           ELSE  // 异常状态处理
               #状态 := 0;  // 恢复到停止状态
               #上阀控制 := FALSE;
               #下阀控制 := FALSE;
       END_CASE;

       // 更新输出状态
       #当前状态 := #状态;
END_FUNCTION_BLOCK

FUNCTION_BLOCK "四参数辅助"   // FB42, SCL
{ S7_Optimized_Access := 'TRUE' }
VERSION : 0.1
// stored: AutoNumber true, IsIECCheckEnabled false, IsRetainMemResEnabled false, MemoryReserve 100, SetENOAutomatically false, UDAEnableTagReadback false
   VAR_INPUT
      启动送风机 : Bool;   // 启动送风机命令
      关闭送风机 : Bool;   // 关闭送风机命令
      设定送风流量 : Real;   // 送风流量设定值
      实际送风流量 : Real;   // 流量变送器测量的实际流量
      流量上阈值 : Real := 10.0;   // 合格区间上限偏差值
      流量下阈值 : Real := 5.0;   // 合格区间下限偏差值
   END_VAR
   VAR_IN_OUT
      调节单元 : Real := 4.0;   // 频率调节单元 4Hz/时间
      调节时间 : Real := 30.0;   // 时间为秒
      调节时间PV : Real;
      变频器频率设定 : Real;   // 输出到变频器的频率设定
   END_VAR
   VAR
      运行状态 : Int := 0;   // 0: 停止, 1: 启动中, 2: 运行中, 3: 关闭中
      起始频率 : Real := 10.0;   // 起始频率10Hz
      最高频率 : Real := 50.0;   // 最高频率50Hz
      频率设定值 : Real := 0.0;   // 内部频率设定值
      流量合格 : Bool := FALSE;   // 流量是否在合格区间内
      TON1 : TON_TIME;
   END_VAR
BEGIN

       // 判断流量是否在合格区间内
       #流量合格 := (#实际送风流量 >= (#设定送风流量 - #流量下阈值)) AND
       (#实际送风流量 <= (#设定送风流量 + #流量上阈值));

       // 状态机
       CASE #运行状态 OF
           0:  // 停止状态
               IF #启动送风机 THEN
                   #运行状态 := 1;  // 转到启动状态
                   #频率设定值 := #起始频率;
                  // #送风机运行 := TRUE;
               END_IF;

           1:  // 启动状态
               IF #关闭送风机 THEN
                   #运行状态 := 3;  // 收到关闭命令，转到关闭状态
               ELSIF #流量合格 THEN
                   #运行状态 := 2;  // 流量达到合格区间，转到运行状态
               ELSIF #TON1.Q THEN
                   // 每分钟调整，最多增减4Hz
                   IF #实际送风流量 < #设定送风流量 - #流量下阈值 THEN
                       // 流量不足，增加频率
                       #频率设定值 := #频率设定值 + #调节单元;
                       IF #频率设定值 > #最高频率 THEN
                           #频率设定值 := #最高频率;
                       END_IF;
                   ELSIF #实际送风流量 > #设定送风流量 + #流量上阈值 THEN
                       // 流量过大，减少频率
                       #频率设定值 := #频率设定值 - #调节单元;
                       IF #频率设定值 < #起始频率 THEN
                           #频率设定值 := #起始频率;
                       END_IF;
                   END_IF;
               END_IF;

           2:  // 运行状态（流量稳定）
               IF #关闭送风机 THEN
                   #运行状态 := 3;  // 收到关闭命令，转到关闭状态
               ELSIF NOT #流量合格 AND #TON1.Q THEN
                   #运行状态 := 1;  // 流量不再合格，转回启动状态继续调节
               END_IF;

           3:  // 关闭状态
               IF #TON1.Q THEN
                   // 每分钟减少4Hz
                   #频率设定值 := #频率设定值 - #调节单元;

                   // 频率低于10Hz时关闭送风机
                   IF #频率设定值 < #起始频率 THEN
                     //  #送风机运行 := FALSE;
                       #频率设定值 := #起始频率;
                       #运行状态 := 0;  // 回到停止状态
                   END_IF;
               END_IF;
       END_CASE;

       #TON1(IN:=NOT #TON1.Q,
             PT:=DINT_TO_TIME(REAL_TO_DINT(#调节时间*1000)));

       #调节时间PV:=DINT_TO_REAL(TIME_TO_DINT(#TON1.ET))*1000;
       // 输出频率设定值
       #变频器频率设定 := #频率设定值;
END_FUNCTION_BLOCK

FUNCTION_BLOCK "闭式保压块"   // FB27, SCL
{ S7_Optimized_Access := 'TRUE' }
VERSION : 0.1
// stored: AutoNumber true, IsIECCheckEnabled false, IsRetainMemResEnabled false, MemoryReserve 100, SetENOAutomatically false, UDAEnableTagReadback false
   VAR_OUTPUT
      MBY等待保压 : Bool;
      MBY正在充气 : Bool;
      MBY保压不佳 : Bool;
      MBY正在保压 : Bool;
      MBY保压正常 : Bool;
   END_VAR
   VAR_IN_OUT
      模式设定 : Real;
      MBY保压 : Bool;
      MQT其他阀 : Bool;
      MCQ充气阀 : Bool;
      MCZ重置 : Bool;
      当前阶段 : Int;
      SV保压低设定 : Real;
      SV保压高设定 : Real;
      SV保压差值 : Real;
      SV保压时 : UInt;
      SV保压分 : UInt;
      SV保压秒 : UInt;
      PV塔内压力 { ExternalAccessible := 'False'; ExternalVisible := 'False'; ExternalWritable := 'False'} : Real;
      PV保压前 { ExternalAccessible := 'False'; ExternalVisible := 'False'; ExternalWritable := 'False'} : Real;
      PV保压后 { ExternalAccessible := 'False'; ExternalVisible := 'False'; ExternalWritable := 'False'} : Real;
      PV保压当前差值 { ExternalAccessible := 'False'; ExternalVisible := 'False'; ExternalWritable := 'False'} : Real;
      PV保压时 { ExternalAccessible := 'False'; ExternalVisible := 'False'; ExternalWritable := 'False'} : UInt;
      PV保压分 { ExternalAccessible := 'False'; ExternalVisible := 'False'; ExternalWritable := 'False'} : UInt;
      PV保压秒 { ExternalAccessible := 'False'; ExternalVisible := 'False'; ExternalWritable := 'False'} : UInt;
   END_VAR
   VAR
      T_1HZ { S7_SetPoint := 'True'} : TON_TIME;
      RT1 { S7_SetPoint := 'True'} : R_TRIG;
   END_VAR
BEGIN
   IF #模式设定 = 1.0 OR #模式设定 = 2.0  THEN

       #RT1(CLK := #MBY保压);
       IF #RT1.Q THEN
           #当前阶段 := 1;
       END_IF;
       IF #MBY保压 THEN
           IF #当前阶段 = 5 THEN
               #当前阶段 := 1;
           END_IF;
      ELSE
           #当前阶段 := 5; 
       END_IF;



       CASE #当前阶段 OF
           1://开始充气
               #MQT其他阀 := 0;
               #MCQ充气阀 := 1;
               #MBY等待保压 := 0;
               #MBY正在充气 := 1;
               #MBY保压不佳 := 0;
               #MBY正在保压 := 0;
               #MBY保压正常 := 0;

               IF (#PV塔内压力 >= #SV保压低设定) AND (#PV塔内压力 <= #SV保压高设定) THEN
                   #MCQ充气阀 := 0;
                   #PV保压前 := #PV塔内压力;
                   #当前阶段 := 2;
               END_IF;
           2://时间记录
               #MQT其他阀 := 0;
               #MCQ充气阀 := 0;
               IF #T_1HZ.Q THEN
                   #PV保压秒 += 1;
                   IF #PV保压秒 >= 60 THEN
                       #PV保压分 += 1;
                       #PV保压秒 := 0;
                       IF #PV保压分 >= 60 THEN
                           #PV保压时 += 1;
                           #PV保压分 := 0;
                       END_IF;
                   END_IF;
               END_IF;
               IF (#PV保压时 > #SV保压时) OR ((#PV保压时 = #SV保压时) AND (#PV保压分 > #SV保压分)) OR ((#PV保压时 = #SV保压时) AND (#PV保压分 = #SV保压分) AND (#PV保压秒 >= #SV保压秒)) THEN
                   #PV保压后 := #PV塔内压力;
                   #当前阶段 := 3;
               END_IF;

               #MBY等待保压 := 0;
               #MBY正在充气 := 0;
               #MBY保压不佳 := 0;
               #MBY正在保压 := 1;
               #MBY保压正常 := 0;

           3://保压结束
               #PV保压当前差值 := ABS(#PV保压前 - #PV保压后);
               #MBY保压正常 := #PV保压当前差值 < #SV保压差值;
               #MBY保压不佳 := NOT (#PV保压当前差值 < #SV保压差值);
               IF #MBY保压正常 OR #MBY保压不佳 THEN
                   #MBY正在保压 := 0;
                   #当前阶段 :=4;
               END_IF;
           4://停止保压，并记录数据



               #MBY正在充气 := 0;

               #MBY正在保压 := 0;



           5://清空数据
               #MCQ充气阀 := 0;
               #MBY保压 := 0;
               #PV保压前 := 0;
               #PV保压后 := 0;
               #PV保压时 := 0;
               #PV保压分 := 0;
               #PV保压秒 := 0;


               #MBY等待保压 := 1;
               #MBY正在充气 := 0;

               #MBY正在保压 := 0;
               #MBY保压正常 := 0;
               #MBY保压不佳 := 0;

               #PV保压当前差值 := 0.0;
       END_CASE;

      (* IF #MCZ重置 THEN
           #当前阶段 := 5;
           #MCZ重置 := FALSE;
       END_IF; *)


       #T_1HZ(IN := NOT #T_1HZ.Q,
              PT := T#1S);
   END_IF;
END_FUNCTION_BLOCK

FUNCTION_BLOCK "A14-阀反馈报警"   // FB20, SCL
{ S7_Optimized_Access := 'TRUE' }
VERSION : 0.1
// stored: AutoNumber true, IsIECCheckEnabled false, IsRetainMemResEnabled false, MemoryReserve 100, SetENOAutomatically false, UDAEnableTagReadback false
   VAR
      补氮阀 : "A8-阀开关报警";
      进氮阀 : "A8-阀开关报警";
      泄压阀 : "A8-阀开关报警";
      气流雾化阀 : "A8-阀开关报警";
      输送进风阀 : "A8-阀开关报警";
      开式排风隔断阀 : "A8-阀开关报警";
      闭式排风隔断阀 : "A8-阀开关报警";
      开式进风隔断阀 : "A8-阀开关报警";
      闭式进风隔断阀 : "A8-阀开关报警";
      一级冷却水阀 : "A8-阀开关报警";
      二级冷冻水阀 : "A8-阀开关报警";
      一级排液阀 : "A8-阀开关报警";
      二级排液阀 : "A8-阀开关报警";
      除雾排液阀 : "A8-阀开关报警";
      溶剂回收排放阀 : "A8-阀开关报警";
      进风冷却水阀 : "A8-阀开关报警";
      塔顶清洗球阀 : "A8-阀开关报警";
      清洗伸缩气缸 : "A8-阀开关报警";
      "71阀开关报警_Instance" { S7_SetPoint := 'True'} : "A8-阀开关报警";
      "71阀开关报警_Instance_1" { S7_SetPoint := 'True'} : "A8-阀开关报警";
   END_VAR
BEGIN

   #补氮阀(阀开报警 => "ABD补氮阀开报警",
        阀关报警 => "ABD补氮阀关报警",
        阀状态 :="QBD补氮阀",
        阀开信号 := "IBD补氮阀开反馈",
        阀关信号 := "IBD补氮阀关反馈");

   #进氮阀(阀开报警 => "AJD进氮阀开报警",
        阀关报警 => "AJD进氮阀关报警",
        阀状态 := "QJD进氮阀",
        阀开信号 := "IJD进氮阀开反馈",
        阀关信号 := "IJD进氮阀关反馈");


   #泄压阀(阀开报警 => "AXY泄压阀开报警",
        阀关报警 => "AXY泄压阀关报警",
        阀状态 := "QXY泄压阀",
        阀开信号 := "IXY泄压阀开反馈",
        阀关信号 := "IXY泄压阀关反馈");

   #气流雾化阀(阀开报警 => "AQL气流雾化阀开报警",
          阀关报警 => "AQL气流雾化阀关报警",
          阀状态 := "QQL气流雾化阀",
          阀开信号 := "IQL气流雾化阀开反馈",
          阀关信号 := "IQL气流雾化阀关反馈");

   #输送进风阀(阀开报警 => "ASS输送进风阀开报警",
          阀关报警 => "ASS输送进风阀关报警",
          阀状态 := "QSS输送进风阀",
          阀开信号 := "ISF输送进风阀开反馈",
          阀关信号 := "ISF输送进风阀关反馈");


   #开式排风隔断阀(阀开报警 => "AKS开式排风隔断阀开报警",
            阀关报警 => "AKS开式排风隔断阀关报警",
            阀状态 := "QKS开式排风隔断阀",
            阀开信号 := "IKS开式排风隔断阀开反馈",
            阀关信号 := "IKS开式排风隔断阀关反馈");

   #闭式排风隔断阀(阀开报警 => "ABS闭式排风隔断阀开报警",
            阀关报警 => "ABS闭式排风隔断阀关报警",
            阀状态 := "QBS闭式排风隔断阀",
            阀开信号 := "IBS闭式排风隔断阀开反馈",
            阀关信号 := "IBS闭式排风隔断阀关反馈");


   #开式进风隔断阀(阀开报警 => "AKS开式进风隔断阀开报警",
            阀关报警 => "AKS开式进风隔断阀关报警",
            阀状态 := "QKS开式进风隔断阀",
            阀开信号 := "IKS开式进风隔断阀开反馈",
            阀关信号 := "IKS开式进风隔断阀关反馈");

   #闭式进风隔断阀(阀开报警 => "ABS闭式进风隔断阀开报警",
            阀关报警 => "ABS闭式进风隔断阀关报警",
            阀状态 := "QBS闭式进风隔断阀",
            阀开信号 := "IBS闭式进风隔断阀开反馈",
            阀关信号 := "IBS闭式进风隔断阀关反馈");

   #一级冷却水阀(阀开报警 => "AYJ一级冷却水阀开报警",
           阀关报警 => "AYJ一级冷却水阀关报警",
           阀状态 := "QYJ一级冷却水阀",
           阀开信号 := "IYJ一级冷却水阀开反馈",
           阀关信号 := "IYJ一级冷却水阀关反馈");


   #二级冷冻水阀(阀开报警 => "AEJ二级冷冻水阀开报警",
           阀关报警 => "AEJ二级冷冻水阀关报警",
           阀状态 := "QEJ二级冷冻水阀",
           阀开信号 := "IEJ二级冷冻水阀开反馈",
           阀关信号 := "IEJ二级冷冻水阀关反馈");

   #一级排液阀(阀开报警 => "AYJ一级排液阀开报警",
          阀关报警 => "AYJ一级排液阀关报警",
          阀状态 := "QYJ一级排液阀",
          阀开信号 := "IYJ一级排液阀开反馈",
          阀关信号 := "IYJ一级排液阀关反馈");


   #二级排液阀(阀开报警 => "AEJ二级排液阀开报警",
          阀关报警 => "AEJ二级排液阀关报警",
          阀状态 := "QEJ二级排液阀",
          阀开信号 := "IEJ二级排液阀开反馈",
          阀关信号 := "IEJ二级排液阀关反馈");

   #除雾排液阀(阀开报警 => "ACW除雾排液阀开报警",
          阀关报警 => "ACW除雾排液阀关报警",
          阀状态 := "QCW除雾排液阀",
          阀开信号 := "ICW除雾排液阀开反馈",
          阀关信号 := "ICW除雾排液阀关反馈");

   #溶剂回收排放阀(阀开报警 => "ARJ溶剂回收排放阀开报警",
            阀关报警 => "ARJ溶剂回收排放阀关报警",
            阀状态 := "QRJ溶剂回收排放阀",
            阀开信号 := "IRJ溶剂回收排放阀开反馈",
            阀关信号 := "IRJ溶剂回收排放阀关反馈");


   #进风冷却水阀(阀开报警 => "AJF进风冷却水阀开报警",
           阀关报警 => "AJF进风冷却水阀关报警",
           阀状态 := "QJF进风冷却水阀",
           阀开信号 := "IJF进风冷却水阀开反馈",
           阀关信号 := "IJF进风冷却水阀关反馈");

   #塔顶清洗球阀(阀开报警 => "ATD塔顶清洗球阀开报警",
           阀关报警 => "ATD塔顶清洗球阀关报警",
           阀状态 := "QTD塔顶清洗球阀",
           阀开信号 := "ITD塔顶清洗球阀开反馈",
           阀关信号 := "ITD塔顶清洗球阀关反馈");


   (* #清洗伸缩气缸(阀开报警 => "AQX清洗伸缩气缸开报警",
           阀关报警 => "AQX清洗伸缩气缸关报警",
           阀状态 := "QQG气缸升降阀",
           阀开信号 := "IQX清洗伸缩气缸开反馈",
           阀关信号 := "IQX清洗伸缩气缸关反馈"); *)
END_FUNCTION_BLOCK

FUNCTION_BLOCK "D3-布袋记录"   // FB74, SCL
{ S7_Optimized_Access := 'TRUE' }
VERSION : 0.1
// stored: AutoNumber true, IsIECCheckEnabled false, IsRetainMemResEnabled false, MemoryReserve 100, SetENOAutomatically false, UDAEnableTagReadback false
   VAR_INPUT
      事件触发器 : Bool;
      清除日志 : Bool;
   END_VAR
   VAR_IN_OUT
      事件记录 : Array[1..20] of String[20];
      事件编号 : Array[1..20] of Int;
      当前记录次数 : Int;
   END_VAR
   VAR
      R_TRIG_Instance { S7_SetPoint := 'True'} : R_TRIG;
      tm_DTL { ExternalAccessible := 'False'; ExternalVisible := 'False'; ExternalWritable := 'False'} : DTL;
   END_VAR
   VAR_TEMP
      tm_Ret : Int;
      tm_i : Int;
      tm_str : String[20];
      tm_year : String[5];
      tm_month : String[3];
      tm_day : String[3];
      tm_hour : String[3];
      tm_minute : String[3];
      tm_second : String[3];
      tm_strcount : String[5];
      tm_strC : String[4];
      tm_empty : Array[1..20] of String[20];
      tm_cempty : Array[1..20] of Int;
   END_VAR
BEGIN
   #R_TRIG_Instance(CLK:=#事件触发器);
   IF #当前记录次数 < 1 THEN
       #当前记录次数 := 1;
   END_IF;

   IF (#当前记录次数 > 9999) OR  #清除日志 THEN
       #当前记录次数 := 1;

       #事件记录 := #tm_empty;
       #事件编号 := #tm_cempty;
       #当前记录次数 := 1;
   END_IF;

   IF #R_TRIG_Instance.Q THEN
       #tm_Ret := RD_LOC_T(#tm_DTL);
       #tm_year := UINT_TO_STRING(#tm_DTL.YEAR);
       #tm_month := USINT_TO_STRING(#tm_DTL.MONTH);
       #tm_day := USINT_TO_STRING(#tm_DTL.DAY);
       #tm_hour := USINT_TO_STRING(#tm_DTL.HOUR+7);
       #tm_minute := USINT_TO_STRING(#tm_DTL.MINUTE);
       #tm_second := USINT_TO_STRING(#tm_DTL.SECOND);
       #tm_str := '';
       #tm_str[1] := #tm_year[2];
       #tm_str[2] := #tm_year[3];
       #tm_str[3] := #tm_year[4];
       #tm_str[4] := #tm_year[5];
       #tm_str[5] := '-';
       IF LEN(#tm_month) = 3 THEN
           #tm_str[6] := #tm_month[2];
           #tm_str[7] := #tm_month[3];
       ELSE
           #tm_str[6] := '0';
           #tm_str[7] := #tm_month[2];
       END_IF;
       #tm_str[8] := '-';
       IF LEN(#tm_day)= 3 THEN
       #tm_str[9] := #tm_day[2];
       #tm_str[10] := #tm_day[3];
   ELSE
       #tm_str[9] := '0';
       #tm_str[10] := #tm_day[2];;
   END_IF;

   #tm_str[11] := ' ';
   IF LEN(#tm_hour) = 3 THEN
       #tm_str[12] := #tm_hour[2];
       #tm_str[13] := #tm_hour[3];
   ELSE
       #tm_str[12] := '0';
       #tm_str[13] := #tm_hour[2];
   END_IF;
   #tm_str[14] := ':';
   IF LEN(#tm_minute) = 3 THEN
       #tm_str[15] := #tm_minute[2];
       #tm_str[16] := #tm_minute[3];
   ELSE
       #tm_str[15] := '0';
       #tm_str[16] := #tm_minute[2];
   END_IF;
       #tm_str[17] := ':';
       IF LEN(#tm_second) = 3 THEN
           #tm_str[18] := #tm_second[2];
           #tm_str[19] := #tm_second[3];
       ELSE
           #tm_str[18] := '0';
           #tm_str[19] := #tm_second[2];
       END_IF;
       #tm_strcount := INT_TO_STRING(#当前记录次数);
       IF LEN(#tm_strcount) = 2 THEN
           #tm_strC[1] := '0';
           #tm_strC[2] := '0';
           #tm_strC[3] := '0';
           #tm_strC[4] := #tm_strcount[2];
       END_IF;

       IF LEN(#tm_strcount) = 3 THEN
           #tm_strC[1] := '0';
           #tm_strC[2] := '0';
           #tm_strC[3] := #tm_strcount[2];
           #tm_strC[4] := #tm_strcount[3];
       END_IF;
       IF LEN(#tm_strcount) = 4 THEN
           #tm_strC[1] := '0';
           #tm_strC[2] := #tm_strcount[2];
           #tm_strC[3] := #tm_strcount[3];
           #tm_strC[4] := #tm_strcount[4];
       END_IF;
       IF LEN(#tm_strcount) =5 THEN
           #tm_strC[1] := #tm_strcount[2];
           #tm_strC[2] := #tm_strcount[3];
           #tm_strC[3] := #tm_strcount[4];
           #tm_strC[4] := #tm_strcount[5];
       END_IF;



       IF #当前记录次数 < 20 THEN
           #事件记录[#当前记录次数] := #tm_str;
           #事件编号[#当前记录次数] :=#当前记录次数;
       ELSE
           FOR #tm_i := 1 TO 19 DO
               #事件编号[#tm_i] := #事件编号[#tm_i + 1];
               #事件编号[#tm_i] := #事件编号[#tm_i + 1];
           END_FOR;
           #事件记录[20] := #tm_str;
           #事件编号[20] := #当前记录次数;
       END_IF;
       #当前记录次数 := #当前记录次数 + 1;
   END_IF;
END_FUNCTION_BLOCK

FUNCTION_BLOCK "12放空阀"   // FB8, SCL
{ S7_Optimized_Access := 'FALSE' }
VERSION : 0.1
// stored: AutoNumber true, IsIECCheckEnabled false, SetENOAutomatically false, UDAEnableTagReadback false
   VAR_INPUT
      条件1 : Real;
      工程上限 : Real;
      工程下限 : Real;
      模拟高限 : Int;
      模拟低限 : Int;
   END_VAR
   VAR_IN_OUT
      模式设定 : Real;
      阀门启动 : Bool;
      阀门输出 : Bool;
      百分比设定值 : Real;
      输出百分比 : Int;
      PID反馈模拟量 : Int;
      YS映射到阀开度 : Real;
   END_VAR
   VAR DB_SPECIFIC
      动画 : Int;
      ST1 : Real;
   END_VAR
   VAR_TEMP
      TEMP_1 : Int;
   END_VAR
BEGIN
   // "IEC_Timer_0_DB".TON(IN:=#输出电源开,
   //                      PT:=T#10s,
   //                      Q=>  #阀开报警检测位);
   // IF #阀开报警检测位 AND #阀开信号  THEN
   //     #阀开异常报警 := TRUE;
   // ELSE
   //     #阀开异常报警 := FALSE;
   // END_IF;
   // "IEC_Timer_0_DB_1".TON (IN:=NOT #输出电源开,
   //                        PT:=T#10s,
   //                        Q=>#阀关报警检测位);
   // IF #阀关报警检测位 AND #阀关信号  THEN
   //     #阀关异常报警 := TRUE; ELSE
   //     #阀关异常报警 :=FALSE;
   // END_IF;
   //手动控制--------------------------------------------------------------------------------------------------------------
   IF #模式设定 = 2.0 THEN

       IF #阀门启动 THEN
           #阀门输出 := TRUE;
           #输出百分比 := REAL_TO_INT((#百分比设定值 - #工程下限) * (#模拟高限 - #模拟低限) / (#工程上限 - #工程下限) + #模拟低限);

       END_IF;
       IF NOT #阀门启动 THEN
           #阀门输出 := FALSE;
           #输出百分比 := REAL_TO_INT(#工程下限);

       END_IF;

   END_IF;

   // 自动启动--------------------------------------------------------------------------------------------------------------
   IF #阀门输出 AND #模式设定 = 1.0 THEN
       (* #输出百分比 := REAL_TO_INT((#百分比设定值 - #工程下限) * (#模拟高限 - #模拟低限) / (#工程上限 - #工程下限) + #模拟低限); *)


       #ST1 := NORM_X_REAL(MIN := 5530, VALUE := #输出百分比, MAX := 27648);
       #YS映射到阀开度 := SCALE_X_REAL(MIN := 0, VALUE := #ST1, MAX := 100);


   END_IF;
   IF NOT #阀门输出 THEN
       #YS映射到阀开度 := 0;
   END_IF;




   (* #TON1(IN := #电机输出 AND #电机电流 < 10,
                          PT := T#60s,
                          Q => #P1);

   IF #P1 OR #电机报警信号 THEN
       #电机报警输出 := TRUE;
   ELSE
       #电机报警输出 := FALSE;
   END_IF; *)



   IF #阀门输出  THEN
       IF "Clock_1Hz" THEN
           #TEMP_1 := #TEMP_1 + 1;
       END_IF;

       IF #TEMP_1 >= 3 THEN
           #TEMP_1 := 0;
       END_IF;
       IF #TEMP_1 < 1 THEN
           #动画 := 0;
       ELSE
           #动画 := 1;
       END_IF;

   END_IF;
   IF NOT #阀门输出 THEN
       #动画 := 0;
   END_IF;




   // IF #阀开异常报警 THEN
   //     #输出电源开 := FALSE;
   // END_IF;
   // IF #阀关异常报警 THEN
   //     #输出电源开 := TRUE;
   // END_IF;
END_FUNCTION_BLOCK

FUNCTION_BLOCK "21模拟量输入"   // FB2, SCL
{ S7_Optimized_Access := 'TRUE' }
VERSION : 0.1
// stored: AutoNumber true, IsIECCheckEnabled false, IsRetainMemResEnabled false, MemoryReserve 100, SetENOAutomatically false, UDAEnableTagReadback false
   VAR_INPUT
      HMI上限 : Real;
      HMI下限 : Real;
      PLC上限 : Int := 27648;
      PLC下限 : Int;
   END_VAR
   VAR_IN_OUT
      "PLC-仪表" : Int;
      HMI仪表 : Real;
   END_VAR
   VAR
      DBD28 : Real;
   END_VAR
BEGIN
   #DBD28 := NORM_X_REAL(MIN := #PLC下限, VALUE := #"PLC-仪表", MAX := #PLC上限);
   #HMI仪表 := SCALE_X_REAL(MIN := #HMI下限, VALUE := #DBD28, MAX := #HMI上限);
END_FUNCTION_BLOCK

FUNCTION_BLOCK "22模拟量输入修正"   // FB10, SCL
{ S7_Optimized_Access := 'TRUE' }
VERSION : 0.1
// stored: AutoNumber true, IsIECCheckEnabled false, IsRetainMemResEnabled false, MemoryReserve 100, SetENOAutomatically false, UDAEnableTagReadback false
   VAR_INPUT
      设备启动 : Bool;
      HMI上限 : Real;
      HMI下限 : Real;
      PLC上限 : Int := 27648;
      PLC下限 : Int;
   END_VAR
   VAR_IN_OUT
      "PLC-仪表" : Int;
      HMI仪表 : Real;
   END_VAR
   VAR
      DBD1 : Real;
   END_VAR
BEGIN
   IF #设备启动 THEN

   #DBD1 := NORM_X_REAL(MIN := #PLC下限, VALUE := #"PLC-仪表", MAX := #PLC上限);
   #HMI仪表 := SCALE_X_REAL(MIN := #HMI下限, VALUE := #DBD1, MAX := #HMI上限);

   ELSE

       #HMI仪表 := 0;
   END_IF;
END_FUNCTION_BLOCK

FUNCTION_BLOCK "23模拟量输出"   // FB36, SCL
{ S7_Optimized_Access := 'TRUE' }
VERSION : 0.1
// stored: AutoNumber true, IsIECCheckEnabled false, IsRetainMemResEnabled false, MemoryReserve 100, SetENOAutomatically false, UDAEnableTagReadback false
   VAR_INPUT
      HMI上限 : Real;
      HMI下限 : Real;
      PLC上限 : Int;
      PLC下限 : Int;
   END_VAR
   VAR_IN_OUT
      PLC调控 : Int;
      HMI设定 : Real;
   END_VAR
   VAR
      DBD1 : Real;
   END_VAR
BEGIN
   #DBD1 := NORM_X_REAL(MIN := #HMI下限, VALUE := #HMI设定, MAX := #HMI上限);
   #PLC调控 := SCALE_X_INT(MIN := #PLC下限, VALUE := #DBD1, MAX := #PLC上限);
END_FUNCTION_BLOCK

FUNCTION_BLOCK "24模拟量其他"   // FB4, SCL
{ S7_Optimized_Access := 'TRUE' }
VERSION : 0.1
// stored: AutoNumber true, IsIECCheckEnabled false, IsRetainMemResEnabled false, MemoryReserve 100, SetENOAutomatically false, UDAEnableTagReadback false
BEGIN
END_FUNCTION_BLOCK

FUNCTION_BLOCK "30-加热控制"   // FB17, SCL
{ S7_Optimized_Access := 'TRUE' }
VERSION : 0.1
// stored: AutoNumber true, IsIECCheckEnabled false, IsRetainMemResEnabled false, MemoryReserve 100, SetENOAutomatically false, UDAEnableTagReadback false
   VAR_INPUT
      条件1 : Real;
   END_VAR
   VAR_IN_OUT
      模式设定 : Real;
      加热控制按钮 : Bool;
      电力调整器信号 : Bool;
      电力调整器报警 : Bool;
      机械温报警信号 : Bool;
      循环风机反馈 : Real;
      循环风机 : Bool;
      加热输出 : Bool;
      AO : Int;
      安全停机 : Bool;
   END_VAR
BEGIN

   //手动控制--------------------------------------------------------------------------------------------------------------
   IF #模式设定 = 2.0 THEN
       //预热器加热手动控制
       IF #加热控制按钮
           AND #电力调整器报警 = FALSE AND #机械温报警信号 = FALSE AND #循环风机反馈 > 20 AND #循环风机 THEN
           #加热输出 := TRUE;

       ELSE

           #加热输出 := FALSE;

       END_IF;
   END_IF;
   IF #模式设定 = 2.0  THEN
       //预热器加热手动控制
       IF NOT #加热控制按钮 THEN


           #加热输出 := FALSE;

       END_IF;
   END_IF;

   //自动模式
   IF #加热输出 THEN
       #AO := -256;
   END_IF;


   IF NOT #加热输出 THEN
       #AO := 0;
   END_IF;
   IF #电力调整器信号 THEN
       #电力调整器报警 := TRUE;
   ELSE


       #电力调整器报警 := FALSE;
   END_IF;

   IF
       #模式设定 = 1 AND (#电力调整器报警 OR #机械温报警信号) THEN

       #安全停机 := 1;
   END_IF;
END_FUNCTION_BLOCK

FUNCTION_BLOCK "31-温度控制"   // FB21, LAD
{ S7_Optimized_Access := 'FALSE' }
VERSION : 0.1
// stored: AutoNumber true, IsIECCheckEnabled false, SetENOAutomatically false, UDAEnableTagReadback false
   VAR_IN_OUT
      进温设定 : Real;
      加热器开关 : Bool;
      自整定开关 : Bool;
      进温读 : Real;
      出温读 : Real;
      尾温读 : Real;
      进风温度P : Real;
      进风温度I : Real;
      进风温度D : Real;
      JF进风温度写读 : Real;
   END_VAR
   VAR DB_SPECIFIC
      CTU { S7_SetPoint := 'True'} : CTU_INT;
      TEMP { S7_SetPoint := 'True'} : Bool;
      TP : Array[0..40] of Bool;
      T1_PV_读 : Int;
      T2_PV_读 : Int;
      T3_PV_读 : Int;
      T4_PV_读 : Int;
      T5_PV_读 : Int;
      T1_SV_写 : Int;
      T1_P值比对1 : Int;
      T1_P值比对2 : Int;
      ST1 : Real;
      ST2 : Real;
      ST3 : Real;
      ST4 : Real;
      ST5 : Real;
      ST16 : Real;
      ST17 : Real;
      ST18 : Real;
      ST20 : Real;
      ST21 : Real;
      ST22 : Real;
      进温P读 : Int;
      进温I读 : Int;
      进温D读 : Int;
      T1_P_I_D_读 : Array[0..2] of Int;
      IEC_Timer_0_Instance { S7_SetPoint := 'True'} : TON_TIME;
      JF进风温度写读辅 { S7_SetPoint := 'True'} : Int;
      进温AT_写 : Int;
      进温AT_读 : Int;
      自整定开关字 : Int;
      加热器开关字 : Int;
   END_VAR
   VAR
      Modbus_Comm_Load_Instance { S7_SetPoint := 'True'} : Modbus_Comm_Load;
      Modbus_Master { S7_SetPoint := 'True'} : Modbus_Master;
   END_VAR
   VAR_TEMP   // added for the SCL form of the ladder/FBD networks
      _w1 : Bool;
      _w2 : Bool;
      _w3 : Bool;
      _w4 : Bool;
   END_VAR
BEGIN

REGION Network 1
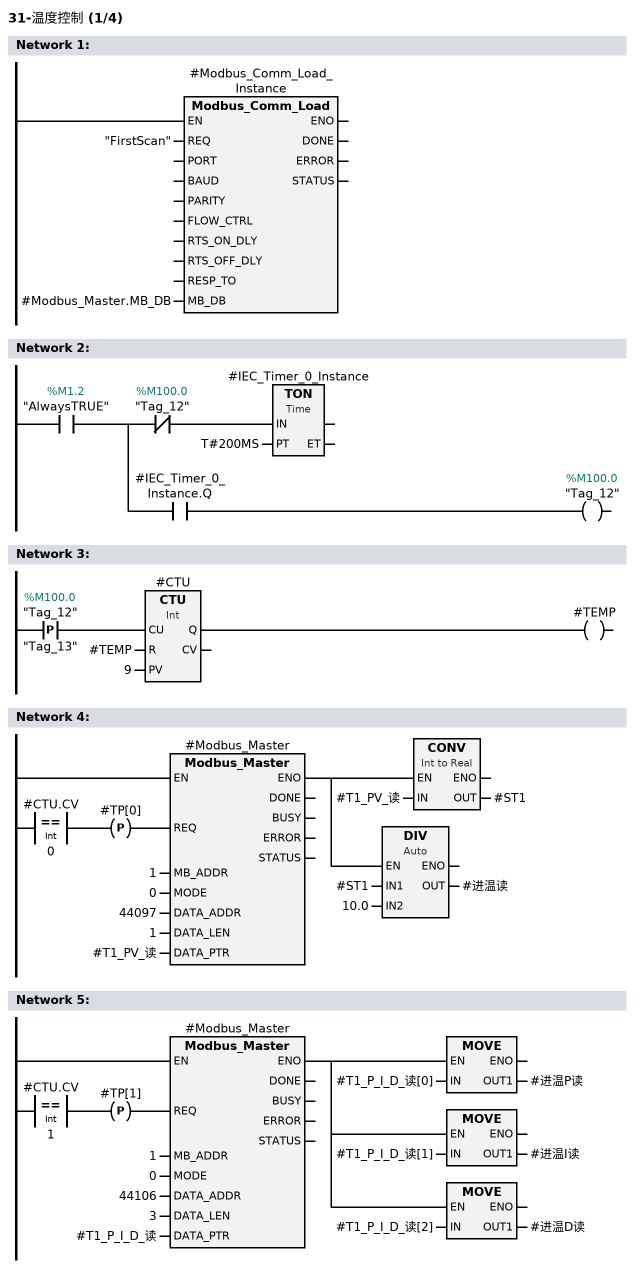
   RUNG wire#powerrail
      #Modbus_Comm_Load_Instance.Modbus_Comm_Load(REQ := "FirstScan", PORT :=, BAUD :=, PARITY :=, FLOW_CTRL :=, RTS_ON_DLY :=, RTS_OFF_DLY :=, RESP_TO :=, MB_DB := #Modbus_Master.MB_DB, DONE =>, ERROR =>, STATUS =>)
   END_RUNG
   // the same network as SCL:
   #Modbus_Comm_Load_Instance(REQ := "FirstScan", MB_DB := #Modbus_Master.MB_DB);   // Modbus_Comm_Load
END_REGION

REGION Network 2
   RUNG wire#powerrail
      Contact( "AlwaysTRUE" )
      wire#w1
      I_Contact( "Tag_12" )
      { S7_Templates := "time_type := Time" } #IEC_Timer_0_Instance.TON(pt := T#200MS, et =>)
   END_RUNG
   RUNG wire#w1
      Contact( #IEC_Timer_0_Instance.Q )
      Coil( "Tag_12" )
   END_RUNG
   // the same network as SCL:
   #IEC_Timer_0_Instance(IN := "AlwaysTRUE" AND NOT "Tag_12", PT := T#200MS);   // TON
   "Tag_12" := "AlwaysTRUE" AND #IEC_Timer_0_Instance.Q;
END_REGION

REGION Network 3
   RUNG wire#powerrail
      P_Contact(operand := "Tag_12", bit := "Tag_13")
      { S7_Templates := "value_type := Int" } #CTU.CTU(r := #TEMP, pv := 9, cv =>)
      Coil( #TEMP )
   END_RUNG
   // the same network as SCL:
   #_w1 := "Tag_12" AND NOT "Tag_13";   // rising edge of "Tag_12"
   "Tag_13" := "Tag_12";
   #CTU(CU := #_w1, R := #TEMP, PV := 9);   // CTU
   #TEMP := #CTU.Q;
END_REGION

REGION Network 4
   RUNG wire#powerrail
      #Modbus_Master.Modbus_Master(REQ := wire#w1, MB_ADDR := 1, MODE := 0, DATA_ADDR := 44097, DATA_LEN := 1, DATA_PTR := #T1_PV_读, DONE =>, BUSY =>, ERROR =>, STATUS =>)
      wire#w2
      { S7_Templates := "[SrcType := Int, DestType := Real]" } Convert(in := #T1_PV_读, out => #ST1)
   END_RUNG
   RUNG wire#powerrail
      { S7_Templates := "SrcType := Int" } EQ_Contact(in1 := #CTU.CV, in2 := 0)
      P_Trig( #TP[0] )
   END_RUNG wire#w1
   RUNG wire#w2
      Div(in1 := #ST1, in2 := 10.0, out => #进温读)
   END_RUNG
   // the same network as SCL:
   #_w1 := #CTU.CV = 0;
   #_w2 := #_w1 AND NOT #TP[0];   // rising edge
   #TP[0] := #_w1;
   #Modbus_Master(REQ := #_w2,   // Modbus_Master
                  MB_ADDR := 1,
                  MODE := 0,
                  DATA_ADDR := 44097,
                  DATA_LEN := 1,
                  DATA_PTR := #T1_PV_读,
                  ENO => #_w3);
   IF #_w3 THEN
       #ST1 := INT_TO_REAL(#T1_PV_读);
       #进温读 := #ST1 / 10.0;
   END_IF;
END_REGION

REGION Network 5
   RUNG wire#powerrail
      #Modbus_Master.Modbus_Master(REQ := wire#w1, MB_ADDR := 1, MODE := 0, DATA_ADDR := 44106, DATA_LEN := 3, DATA_PTR := #T1_P_I_D_读, DONE =>, BUSY =>, ERROR =>, STATUS =>)
      wire#w2
      Move(in := #T1_P_I_D_读[0], out1 => #进温P读)
   END_RUNG
   RUNG wire#powerrail
      { S7_Templates := "SrcType := Int" } EQ_Contact(in1 := #CTU.CV, in2 := 1)
      P_Trig( #TP[1] )
   END_RUNG wire#w1
   RUNG wire#w2
      Move(in := #T1_P_I_D_读[1], out1 => #进温I读)
   END_RUNG
   RUNG wire#w2
      Move(in := #T1_P_I_D_读[2], out1 => #进温D读)
   END_RUNG
   // the same network as SCL:
   #_w1 := #CTU.CV = 1;
   #_w2 := #_w1 AND NOT #TP[1];   // rising edge
   #TP[1] := #_w1;
   #Modbus_Master(REQ := #_w2,   // Modbus_Master
                  MB_ADDR := 1,
                  MODE := 0,
                  DATA_ADDR := 44106,
                  DATA_LEN := 3,
                  DATA_PTR := #T1_P_I_D_读,
                  ENO => #_w3);
   IF #_w3 THEN
       #进温P读 := #T1_P_I_D_读[0];
       #进温I读 := #T1_P_I_D_读[1];
       #进温D读 := #T1_P_I_D_读[2];
   END_IF;
END_REGION

REGION Network 6
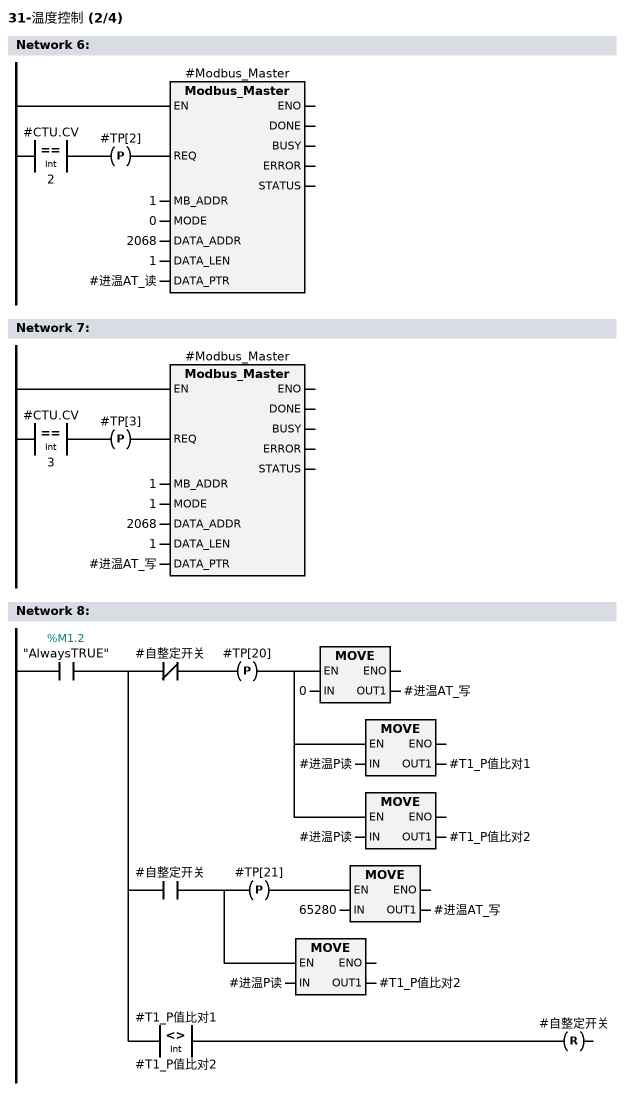
   RUNG wire#powerrail
      #Modbus_Master.Modbus_Master(REQ := wire#w1, MB_ADDR := 1, MODE := 0, DATA_ADDR := 2068, DATA_LEN := 1, DATA_PTR := #进温AT_读, DONE =>, BUSY =>, ERROR =>, STATUS =>)
   END_RUNG
   RUNG wire#powerrail
      { S7_Templates := "SrcType := Int" } EQ_Contact(in1 := #CTU.CV, in2 := 2)
      P_Trig( #TP[2] )
   END_RUNG wire#w1
   // the same network as SCL:
   #_w1 := #CTU.CV = 2;
   #_w2 := #_w1 AND NOT #TP[2];   // rising edge
   #TP[2] := #_w1;
   #Modbus_Master(REQ := #_w2, MB_ADDR := 1, MODE := 0, DATA_ADDR := 2068, DATA_LEN := 1, DATA_PTR := #进温AT_读);   // Modbus_Master
END_REGION

REGION Network 7
   RUNG wire#powerrail
      #Modbus_Master.Modbus_Master(REQ := wire#w1, MB_ADDR := 1, MODE := 1, DATA_ADDR := 2068, DATA_LEN := 1, DATA_PTR := #进温AT_写, DONE =>, BUSY =>, ERROR =>, STATUS =>)
   END_RUNG
   RUNG wire#powerrail
      { S7_Templates := "SrcType := Int" } EQ_Contact(in1 := #CTU.CV, in2 := 3)
      P_Trig( #TP[3] )
   END_RUNG wire#w1
   // the same network as SCL:
   #_w1 := #CTU.CV = 3;
   #_w2 := #_w1 AND NOT #TP[3];   // rising edge
   #TP[3] := #_w1;
   #Modbus_Master(REQ := #_w2, MB_ADDR := 1, MODE := 1, DATA_ADDR := 2068, DATA_LEN := 1, DATA_PTR := #进温AT_写);   // Modbus_Master
END_REGION

REGION Network 8
   RUNG wire#powerrail
      Contact( "AlwaysTRUE" )
      wire#w1
      I_Contact( #自整定开关 )
      P_Trig( #TP[20] )
      wire#w2
      Move(in := 0, out1 => #进温AT_写)
   END_RUNG
   RUNG wire#w2
      Move(in := #进温P读, out1 => #T1_P值比对1)
   END_RUNG
   RUNG wire#w2
      Move(in := #进温P读, out1 => #T1_P值比对2)
   END_RUNG
   RUNG wire#w1
      Contact( #自整定开关 )
      wire#w3
      P_Trig( #TP[21] )
      Move(in := 65280, out1 => #进温AT_写)
   END_RUNG
   RUNG wire#w3
      Move(in := #进温P读, out1 => #T1_P值比对2)
   END_RUNG
   RUNG wire#w1
      { S7_Templates := "SrcType := Int" } NE_Contact(in1 := #T1_P值比对1, in2 := #T1_P值比对2)
      R_Coil( #自整定开关 )
   END_RUNG
   // the same network as SCL:
   #_w1 := "AlwaysTRUE" AND NOT #自整定开关;
   #_w2 := #_w1 AND NOT #TP[20];   // rising edge
   #TP[20] := #_w1;
   IF #_w2 THEN
       #进温AT_写 := 0;
       #T1_P值比对1 := #进温P读;
       #T1_P值比对2 := #进温P读;
   END_IF;
   #_w3 := "AlwaysTRUE" AND #自整定开关;
   #_w4 := #_w3 AND NOT #TP[21];   // rising edge
   #TP[21] := #_w3;
   IF #_w4 THEN #进温AT_写 := 65280; END_IF;
   IF #_w3 THEN #T1_P值比对2 := #进温P读; END_IF;
   IF "AlwaysTRUE" AND (#T1_P值比对1 <> #T1_P值比对2) THEN #自整定开关 := FALSE; END_IF;
END_REGION

REGION Network 9
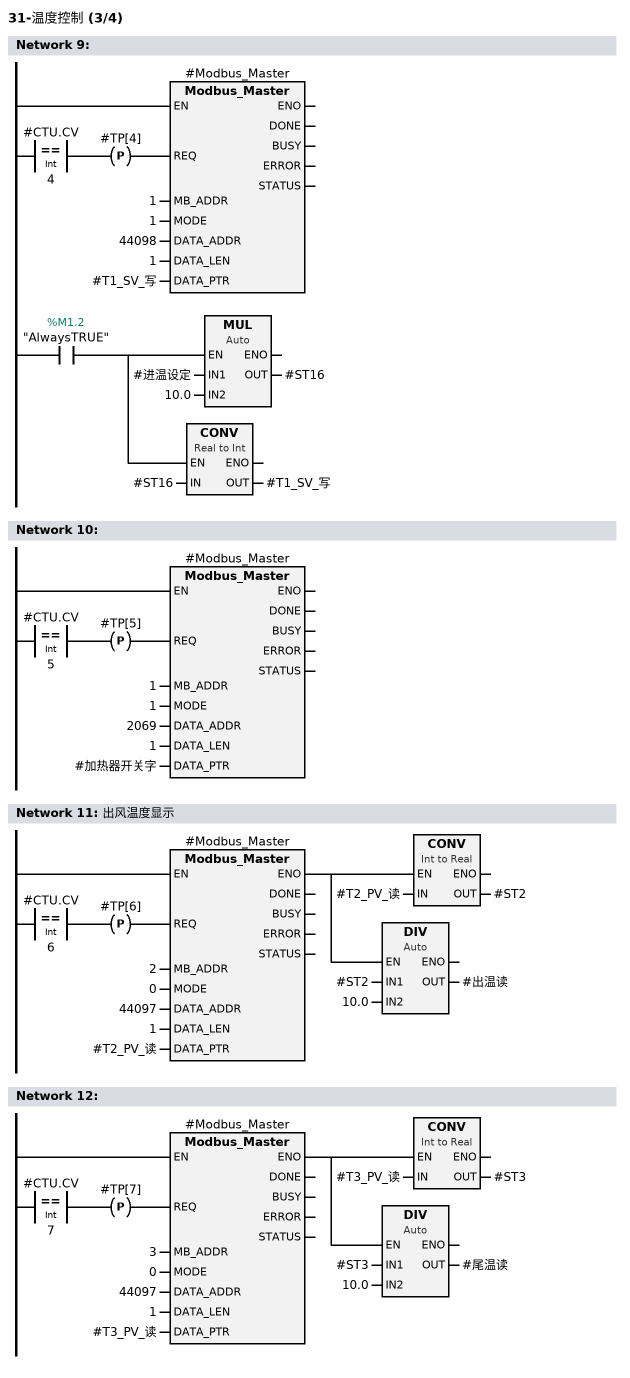
   RUNG wire#powerrail
      #Modbus_Master.Modbus_Master(REQ := wire#w1, MB_ADDR := 1, MODE := 1, DATA_ADDR := 44098, DATA_LEN := 1, DATA_PTR := #T1_SV_写, DONE =>, BUSY =>, ERROR =>, STATUS =>)
   END_RUNG
   RUNG wire#powerrail
      { S7_Templates := "SrcType := Int" } EQ_Contact(in1 := #CTU.CV, in2 := 4)
      P_Trig( #TP[4] )
   END_RUNG wire#w1
   RUNG wire#powerrail
      Contact( "AlwaysTRUE" )
      wire#w2
      Mul(in1 := #进温设定, in2 := 10.0, out => #ST16)
   END_RUNG
   RUNG wire#w2
      { S7_Templates := "[SrcType := Real, DestType := Int]" } Convert(in := #ST16, out => #T1_SV_写)
   END_RUNG
   // the same network as SCL:
   #_w1 := #CTU.CV = 4;
   #_w2 := #_w1 AND NOT #TP[4];   // rising edge
   #TP[4] := #_w1;
   #Modbus_Master(REQ := #_w2, MB_ADDR := 1, MODE := 1, DATA_ADDR := 44098, DATA_LEN := 1, DATA_PTR := #T1_SV_写);   // Modbus_Master
   IF "AlwaysTRUE" THEN
       #ST16 := #进温设定 * 10.0;
       #T1_SV_写 := REAL_TO_INT(#ST16);
   END_IF;
END_REGION

REGION Network 10
   RUNG wire#powerrail
      #Modbus_Master.Modbus_Master(REQ := wire#w1, MB_ADDR := 1, MODE := 1, DATA_ADDR := 2069, DATA_LEN := 1, DATA_PTR := #加热器开关字, DONE =>, BUSY =>, ERROR =>, STATUS =>)
   END_RUNG
   RUNG wire#powerrail
      { S7_Templates := "SrcType := Int" } EQ_Contact(in1 := #CTU.CV, in2 := 5)
      P_Trig( #TP[5] )
   END_RUNG wire#w1
   // the same network as SCL:
   #_w1 := #CTU.CV = 5;
   #_w2 := #_w1 AND NOT #TP[5];   // rising edge
   #TP[5] := #_w1;
   #Modbus_Master(REQ := #_w2, MB_ADDR := 1, MODE := 1, DATA_ADDR := 2069, DATA_LEN := 1, DATA_PTR := #加热器开关字);   // Modbus_Master
END_REGION

REGION Network 11: 出风温度显示
   RUNG wire#powerrail
      #Modbus_Master.Modbus_Master(REQ := wire#w1, MB_ADDR := 2, MODE := 0, DATA_ADDR := 44097, DATA_LEN := 1, DATA_PTR := #T2_PV_读, DONE =>, BUSY =>, ERROR =>, STATUS =>)
      wire#w2
      { S7_Templates := "[SrcType := Int, DestType := Real]" } Convert(in := #T2_PV_读, out => #ST2)
   END_RUNG
   RUNG wire#powerrail
      { S7_Templates := "SrcType := Int" } EQ_Contact(in1 := #CTU.CV, in2 := 6)
      P_Trig( #TP[6] )
   END_RUNG wire#w1
   RUNG wire#w2
      Div(in1 := #ST2, in2 := 10.0, out => #出温读)
   END_RUNG
   // the same network as SCL:
   #_w1 := #CTU.CV = 6;
   #_w2 := #_w1 AND NOT #TP[6];   // rising edge
   #TP[6] := #_w1;
   #Modbus_Master(REQ := #_w2,   // Modbus_Master
                  MB_ADDR := 2,
                  MODE := 0,
                  DATA_ADDR := 44097,
                  DATA_LEN := 1,
                  DATA_PTR := #T2_PV_读,
                  ENO => #_w3);
   IF #_w3 THEN
       #ST2 := INT_TO_REAL(#T2_PV_读);
       #出温读 := #ST2 / 10.0;
   END_IF;
END_REGION

REGION Network 12
   RUNG wire#powerrail
      #Modbus_Master.Modbus_Master(REQ := wire#w1, MB_ADDR := 3, MODE := 0, DATA_ADDR := 44097, DATA_LEN := 1, DATA_PTR := #T3_PV_读, DONE =>, BUSY =>, ERROR =>, STATUS =>)
      wire#w2
      { S7_Templates := "[SrcType := Int, DestType := Real]" } Convert(in := #T3_PV_读, out => #ST3)
   END_RUNG
   RUNG wire#powerrail
      { S7_Templates := "SrcType := Int" } EQ_Contact(in1 := #CTU.CV, in2 := 7)
      P_Trig( #TP[7] )
   END_RUNG wire#w1
   RUNG wire#w2
      Div(in1 := #ST3, in2 := 10.0, out => #尾温读)
   END_RUNG
   // the same network as SCL:
   #_w1 := #CTU.CV = 7;
   #_w2 := #_w1 AND NOT #TP[7];   // rising edge
   #TP[7] := #_w1;
   #Modbus_Master(REQ := #_w2,   // Modbus_Master
                  MB_ADDR := 3,
                  MODE := 0,
                  DATA_ADDR := 44097,
                  DATA_LEN := 1,
                  DATA_PTR := #T3_PV_读,
                  ENO => #_w3);
   IF #_w3 THEN
       #ST3 := INT_TO_REAL(#T3_PV_读);
       #尾温读 := #ST3 / 10.0;
   END_IF;
END_REGION

REGION Network 13
   // 冷水机温du
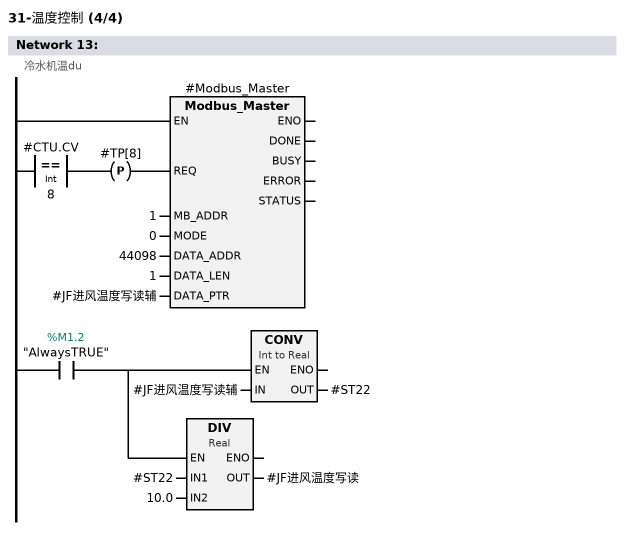
   RUNG wire#powerrail
      #Modbus_Master.Modbus_Master(REQ := wire#w1, MB_ADDR := 1, MODE := 0, DATA_ADDR := 44098, DATA_LEN := 1, DATA_PTR := #JF进风温度写读辅, DONE =>, BUSY =>, ERROR =>, STATUS =>)
   END_RUNG
   RUNG wire#powerrail
      { S7_Templates := "SrcType := Int" } EQ_Contact(in1 := #CTU.CV, in2 := 8)
      P_Trig( #TP[8] )
   END_RUNG wire#w1
   RUNG wire#powerrail
      Contact( "AlwaysTRUE" )
      wire#w2
      { S7_Templates := "[SrcType := Int, DestType := Real]" } Convert(in := #JF进风温度写读辅, out => #ST22)
   END_RUNG
   RUNG wire#w2
      { S7_Templates := "SrcType := Real" } Div(in1 := #ST22, in2 := 10.0, out => #JF进风温度写读)
   END_RUNG
   // the same network as SCL:
   #_w1 := #CTU.CV = 8;
   #_w2 := #_w1 AND NOT #TP[8];   // rising edge
   #TP[8] := #_w1;
   #Modbus_Master(REQ := #_w2,   // Modbus_Master
                  MB_ADDR := 1,
                  MODE := 0,
                  DATA_ADDR := 44098,
                  DATA_LEN := 1,
                  DATA_PTR := #JF进风温度写读辅);
   IF "AlwaysTRUE" THEN
       #ST22 := INT_TO_REAL(#JF进风温度写读辅);
       #JF进风温度写读 := #ST22 / 10.0;
   END_IF;
END_REGION

REGION Network 14 (SCL)
   #进风温度P := INT_TO_REAL(#进温P读);
   #进风温度I := INT_TO_REAL(#进温I读);
   #进风温度D := INT_TO_REAL(#进温D读);
   IF #加热器开关 THEN
       #加热器开关字 := 65280;
   ELSE
       #加热器开关字 := 0;
   END_IF;
END_REGION
END_FUNCTION_BLOCK

FUNCTION_BLOCK "Modbus_Comm_Load"   // FB640, SCL
TITLE = Modbus port configuration
AUTHOR : SIMATIC
FAMILY : MODBUS
NAME : MBCOMLOA
VERSION : 5.0
// stored: IsIECCheckEnabled true, SetENOAutomatically false, UDAEnableTagReadback false
   VAR_INPUT
      REQ : Bool;   // Startet die Konfiguration für Modbus RTU Kommunikation / Activates the configuration for Modbus RTU communication
      PORT : PORT := 0;   // Kommunikationsport, Hardwarekennung / Communication port, Hardware Identifier
      BAUD : UDInt := 9600;   // Datenübertragungsrate / Transmission rate
      PARITY : UInt := 0;   // Parität / Parity
      FLOW_CTRL : UInt := 0;   // Flusskontrolle / Enables or disables flow control
      RTS_ON_DLY : UInt := 0;   // Wartezeit nach Aktivierung von RTS, vor Übertragung von Tx-Daten (ms) / Time to wait after activating RTS before transmission will be initiated
      RTS_OFF_DLY : UInt := 0;   // Wartezeit nach Übertragung von Tx-Daten, bevor RTS deaktiviert wird (ms) / Time to wait before de-activating RTS once transmission has been completed
      RESP_TO : UInt := 1000;   // Zeitdauer, die der Master auf ein Antworttelegramm wartet / Time period that the master waits for a response
   END_VAR
   VAR_OUTPUT
      DONE : Bool;   // Anweisung beendet ohne Fehler / Instruction finished without error
      ERROR : Bool;   // Anweisung beendet mit Fehler / Instruction finished with error
      STATUS : Word := W#16#7000;   // Detailllierte Fehlerinformation / Detailed error information
   END_VAR
   VAR_IN_OUT
      MB_DB : P2P_MB_BASE;   // Zeiger auf den Parameter MB_DB des Modbus_Master oder Modbus_Slave Instanz-DBs / Reference to the parameter MB_DB of Modbus_Master or Modbus_Slave instance DB
   END_VAR
   VAR
      ICHAR_GAP : Word;   // Anzahl der Bitzeiten zwischen den Zeichen / Inter-character gap
      RETRIES : Word;   // Anzahl Wiederholversuche bei Timeout / Number of retries in case of a timeout
      MODE : USInt := 16#00;   // Duplex-Betriebsart / Duplex operation mode
      LINE_PRE : USInt := 16#00;   // Vorbelegung der Empfangsleitung / Presetting of the receive line
      BRK_DET : USInt := 16#00;   // RS232 Break-Erkennung / RS232 BREAK Handling
      EN_DIAG_ALARM : Bool;   // Generierung von Diagnosemeldungen aktivieren / Enable diagnostic alarm generation
      STOP_BITS : USInt := 1;   // Number of STOP bits; 1=1 Stop bit; 2=2 Stop bits
      EN_SUPPLY_VOLT : Bool;   // Diagnose für fehlende Versorgungsspannung L+ einschalten / Enable supply voltage diagnostic
      b_e_REQ : Bool;   // Flankenbit für REQ / Edge flag for REQ
      y_state : SInt := 16#00;   // Status der Anweisung / State of instruction
      Send_Config { S7_SetPoint := 'True'} : Send_Config;   // Lokale Instanz der Anweisung Send_Config / Local instance of the instruction Send_Config
      Receive_Config { S7_SetPoint := 'True'} : Receive_Config;   // Lokale Instanz der Anweisung Receive_Config / Local instance of the instruction Receive_Config
      Receive_Conditions { S7_SetPoint := 'True'} : Receive_Conditions;   // Parameter für Receive_Config / Parameter for Receive_Config
      WRREC { S7_SetPoint := 'True'} : WRREC;   // Lokale Instanz der Anweisung WRREC / Local instance of the instruction WRREC
      RDREC { S7_SetPoint := 'True'} : RDREC;   // Lokale Instanz der Anweisung RDREC / Local instance of the instruction RDREC
      port_w_record { ExternalVisible := 'False'; S7_SetPoint := 'True'} : P2P_MB_PortData;   // Nur für internen Gebrauch / For internal use only
      err_record { ExternalVisible := 'False'; S7_SetPoint := 'True'} : P2P_RdEstat;   // Nur für internen Gebrauch / For internal use only
      ftrs_w_record { ExternalVisible := 'False'; S7_SetPoint := 'True'} : P2P_FeaturesData;   // Nur für internen Gebrauch / For internal use only
   END_VAR
BEGIN
END_FUNCTION_BLOCK

FUNCTION_BLOCK "Send_Config"   // FB611, SCL
TITLE = Send Configuration
AUTHOR : SIMATIC
FAMILY : Freeport
NAME : SendConf
VERSION : 4.0
// stored: IsIECCheckEnabled false, SetENOAutomatically false, UDAEnableTagReadback false
   VAR_INPUT
      REQ : Bool;   // Startet die Konfiguration für Senden bei steigender Flanke / Activates the configuration for sending on rising edge
      PORT : PORT := 0;   // Kommunikationsport, Hardwarekennung / Communication port, Hardware Identifier
      RTSONDLY : UInt := 16#00;   // Wartezeit nach Aktivierung von RTS, vor Übertragung von Tx-Daten (ms) / Time to wait after activating RTS before transmission will be initiated (ms)
      RTSOFFDLY : UInt := 16#00;   // Wartezeit nach Übertragung von Tx-Daten, bevor RTS deaktiviert wird (ms) / Time to wait before de-activating RTS once transmission has been completed (ms)
      BREAK : UInt := 16#00;   // Pause vor Start jeder Übertragung (Bitzeiten) / On start of a message, a break will be sent for the specified no. of bit times
      IDLELINE : UInt := 16#00;   // Leerlaufzeit vor Start jeder Übertragung (Bitzeiten) / Number of bits times the line will be idle before the next transmission
      USR_END : String[2] := '';   // Anzahl der Endekennzeichen / Number of characters in the end delimiter
      APP_END : String[5] := '';   // Anzahl angehängter Zeichen / Number of characters to be appended to the transmitted message
   END_VAR
   VAR_OUTPUT
      DONE : Bool;   // Anweisung beendet ohne Fehler / Instruction finished without error
      ERROR : Bool;   // Anweisung beendet mit Fehler / Instruction finished with error
      STATUS : Word := W#16#7000;   // Zusätzliche Fehlerinformation / Detailed error information
   END_VAR
   VAR
      b_e_REQ : Bool;   // Flankenbit für REQ / Edge flag for REQ
      y_state : SInt := 16#00;   // Status der Anweisung / State of instruction
      WRREC { S7_SetPoint := 'True'} : WRREC;   // Lokale Instanz der Anweisung WRREC / Local instance of instruction WRREC
      RDREC { S7_SetPoint := 'True'} : RDREC;   // Lokale Instanz der Anweisung RDREC / Local instance of instruction RDREC
      w_record { S7_SetPoint := 'True'} : P2P_SendCfgData;   // Nur für internen Gebrauch / For internal use only
      r_record { S7_SetPoint := 'True'} : P2P_RdEstat;   // Nur für internen Gebrauch / For internal use only
   END_VAR
BEGIN
END_FUNCTION_BLOCK

FUNCTION_BLOCK "Receive_Config"   // FB612, SCL
TITLE = Receive Configuration
AUTHOR : SIMATIC
FAMILY : Freeport
NAME : RcvConf
VERSION : 4.0
// stored: IsIECCheckEnabled false, SetENOAutomatically false, UDAEnableTagReadback false
   VAR_INPUT
      REQ : Bool;   // Startet die Konfiguration für Empfangen bei steigender Flanke / Activates the configuration for receiving on rising edge
      PORT : PORT := 0;   // Kommunikationsport, Hardwarekennung / Communication port, Hardware Identifier
      Receive_Conditions : Variant;   // Referenz auf die Empfangsparameter (Receive_Conditions) / Reference to Receive_Conditions
   END_VAR
   VAR_OUTPUT
      DONE : Bool;   // Anweisung beendet ohne Fehler / Instruction finished without error
      ERROR : Bool;   // Anweisung beendet mit Fehler / Instruction finished with error
      STATUS : Word := W#16#7000;   // Zusätzliche Fehlerinformation / Detailed error information
   END_VAR
   VAR
      b_e_REQ : Bool;   // Flankenbit für REQ / Edge flag for REQ
      y_state : SInt := 16#00;   // Status der Anweisung / State of instruction
      WRREC { S7_SetPoint := 'True'} : WRREC;   // Lokale Instanz der Anweisung WRREC / Local instance of instruction WRREC
      RDREC { S7_SetPoint := 'True'} : RDREC;   // Lokale Instanz der Anweisung RDREC / Local instance of instruction RDREC
      w_record { S7_SetPoint := 'True'} : P2P_RcvCfgData;   // Nur für internen Gebrauch / For internal use only
      r_record { S7_SetPoint := 'True'} : P2P_RdEstat;   // Nur für internen Gebrauch / For internal use only
   END_VAR
BEGIN
END_FUNCTION_BLOCK

FUNCTION_BLOCK "32-油炉控制"   // FB22, LAD
{ S7_Optimized_Access := 'FALSE' }
VERSION : 0.1
// stored: AutoNumber true, IsIECCheckEnabled false, SetENOAutomatically false, UDAEnableTagReadback false
   VAR_IN_OUT
      油炉温度写 : Real;
      油炉温度读 : Real;
      油炉循环泵启停 : Bool;
      油炉报警 : Bool;
      油炉冷却阀启停状态 : Bool;
      油炉加热泵启停状态 : Bool;
      油炉加热器1状态 : Bool;
      油炉加热器2状态 : Bool;
      油炉运行状态 : Bool;
      油炉自整定状态 : Bool;
      油炉强制冷却状态 : Bool;
      YL油炉温度写读 : Real;
   END_VAR
   VAR
      MB_COMM_LOAD { S7_SetPoint := 'True'} : Modbus_Comm_Load;
      MB_MASTER_DB { S7_SetPoint := 'True'} : Modbus_Master;
   END_VAR
   VAR DB_SPECIFIC
      CTU { S7_SetPoint := 'True'} : CTU_INT;
      TEMP { S7_SetPoint := 'True'} : Bool;
      TP : Array[0..40] of Bool;
      油炉温度读辅 : Int;
      油炉温度写辅 : Int;
      ST1 : Real;
      ST2 : Real;
      ST3 : Real;
      ST4 : Real;
      ST5 : Real;
      ST16 : Real;
      ST17 : Real;
      ST18 : Real;
      ST20 : Real;
      ST21 : Real;
      ST22 : Real;
      油炉状态1 : Int;
      油炉状态2 : Int;
      油炉启停字 : Int;
      油炉加热状态 : Int;
      油炉运行标志 : Int;
      YL油炉温度写读辅 : Int;
   END_VAR
   VAR
      Modbus_Comm_Load { S7_SetPoint := 'True'} : Modbus_Comm_Load;
      Modbus_Master { S7_SetPoint := 'True'} : Modbus_Master;
   END_VAR
   VAR_TEMP   // added for the SCL form of the ladder/FBD networks
      _w1 : Bool;
      _w2 : Bool;
      _w3 : Bool;
   END_VAR
BEGIN

REGION Network 1
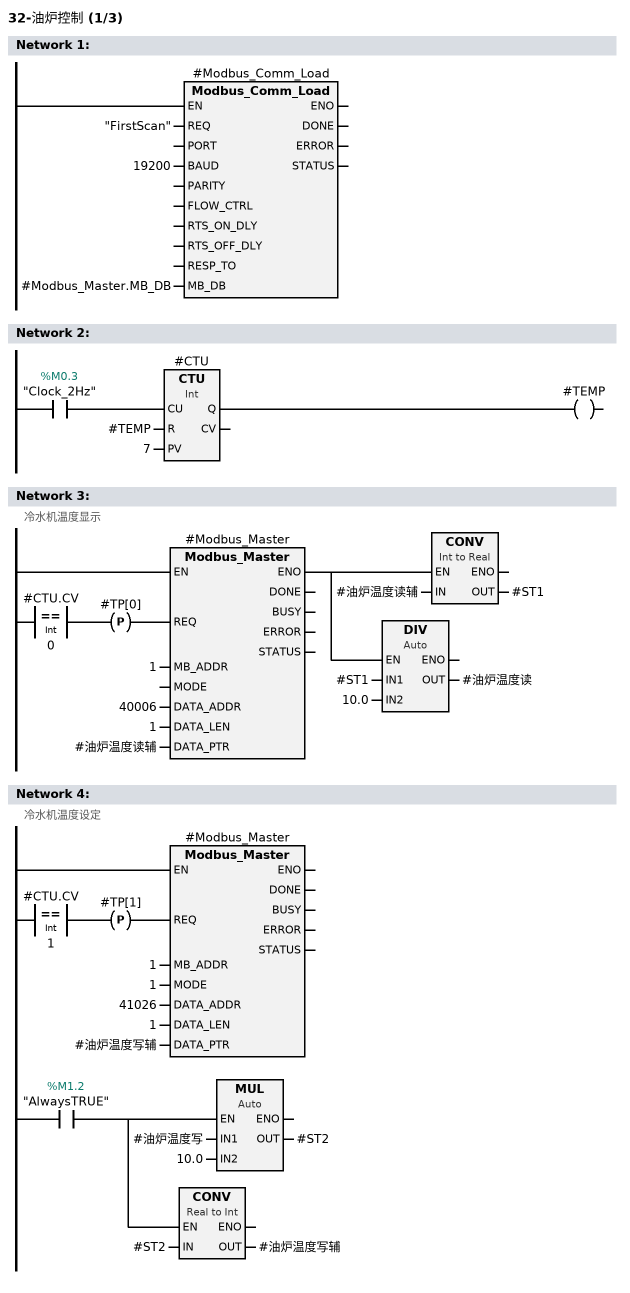
   RUNG wire#powerrail
      #Modbus_Comm_Load.Modbus_Comm_Load(REQ := "FirstScan", PORT :=, BAUD := 19200, PARITY :=, FLOW_CTRL :=, RTS_ON_DLY :=, RTS_OFF_DLY :=, RESP_TO :=, MB_DB := #Modbus_Master.MB_DB, DONE =>, ERROR =>, STATUS =>)
   END_RUNG
   // the same network as SCL:
   #Modbus_Comm_Load(REQ := "FirstScan", BAUD := 19200, MB_DB := #Modbus_Master.MB_DB);   // Modbus_Comm_Load
END_REGION

REGION Network 2
   RUNG wire#powerrail
      Contact( "Clock_2Hz" )
      { S7_Templates := "value_type := Int" } #CTU.CTU(r := #TEMP, pv := 7, cv =>)
      Coil( #TEMP )
   END_RUNG
   // the same network as SCL:
   #CTU(CU := "Clock_2Hz", R := #TEMP, PV := 7);   // CTU
   #TEMP := #CTU.Q;
END_REGION

REGION Network 3
   // 冷水机温度显示
   RUNG wire#powerrail
      #Modbus_Master.Modbus_Master(REQ := wire#w1, MB_ADDR := 1, MODE :=, DATA_ADDR := 40006, DATA_LEN := 1, DATA_PTR := #油炉温度读辅, DONE =>, BUSY =>, ERROR =>, STATUS =>)
      wire#w2
      { S7_Templates := "[SrcType := Int, DestType := Real]" } Convert(in := #油炉温度读辅, out => #ST1)
   END_RUNG
   RUNG wire#powerrail
      { S7_Templates := "SrcType := Int" } EQ_Contact(in1 := #CTU.CV, in2 := 0)
      P_Trig( #TP[0] )
   END_RUNG wire#w1
   RUNG wire#w2
      Div(in1 := #ST1, in2 := 10.0, out => #油炉温度读)
   END_RUNG
   // the same network as SCL:
   #_w1 := #CTU.CV = 0;
   #_w2 := #_w1 AND NOT #TP[0];   // rising edge
   #TP[0] := #_w1;
   #Modbus_Master(REQ := #_w2,   // Modbus_Master
                  MB_ADDR := 1,
                  DATA_ADDR := 40006,
                  DATA_LEN := 1,
                  DATA_PTR := #油炉温度读辅,
                  ENO => #_w3);
   IF #_w3 THEN
       #ST1 := INT_TO_REAL(#油炉温度读辅);
       #油炉温度读 := #ST1 / 10.0;
   END_IF;
END_REGION

REGION Network 4
   // 冷水机温度设定
   RUNG wire#powerrail
      #Modbus_Master.Modbus_Master(REQ := wire#w1, MB_ADDR := 1, MODE := 1, DATA_ADDR := 41026, DATA_LEN := 1, DATA_PTR := #油炉温度写辅, DONE =>, BUSY =>, ERROR =>, STATUS =>)
   END_RUNG
   RUNG wire#powerrail
      { S7_Templates := "SrcType := Int" } EQ_Contact(in1 := #CTU.CV, in2 := 1)
      P_Trig( #TP[1] )
   END_RUNG wire#w1
   RUNG wire#powerrail
      Contact( "AlwaysTRUE" )
      wire#w2
      Mul(in1 := #油炉温度写, in2 := 10.0, out => #ST2)
   END_RUNG
   RUNG wire#w2
      { S7_Templates := "[SrcType := Real, DestType := Int]" } Convert(in := #ST2, out => #油炉温度写辅)
   END_RUNG
   // the same network as SCL:
   #_w1 := #CTU.CV = 1;
   #_w2 := #_w1 AND NOT #TP[1];   // rising edge
   #TP[1] := #_w1;
   #Modbus_Master(REQ := #_w2, MB_ADDR := 1, MODE := 1, DATA_ADDR := 41026, DATA_LEN := 1, DATA_PTR := #油炉温度写辅);   // Modbus_Master
   IF "AlwaysTRUE" THEN
       #ST2 := #油炉温度写 * 10.0;
       #油炉温度写辅 := REAL_TO_INT(#ST2);
   END_IF;
END_REGION

REGION Network 5
   // 冷水机温度设定
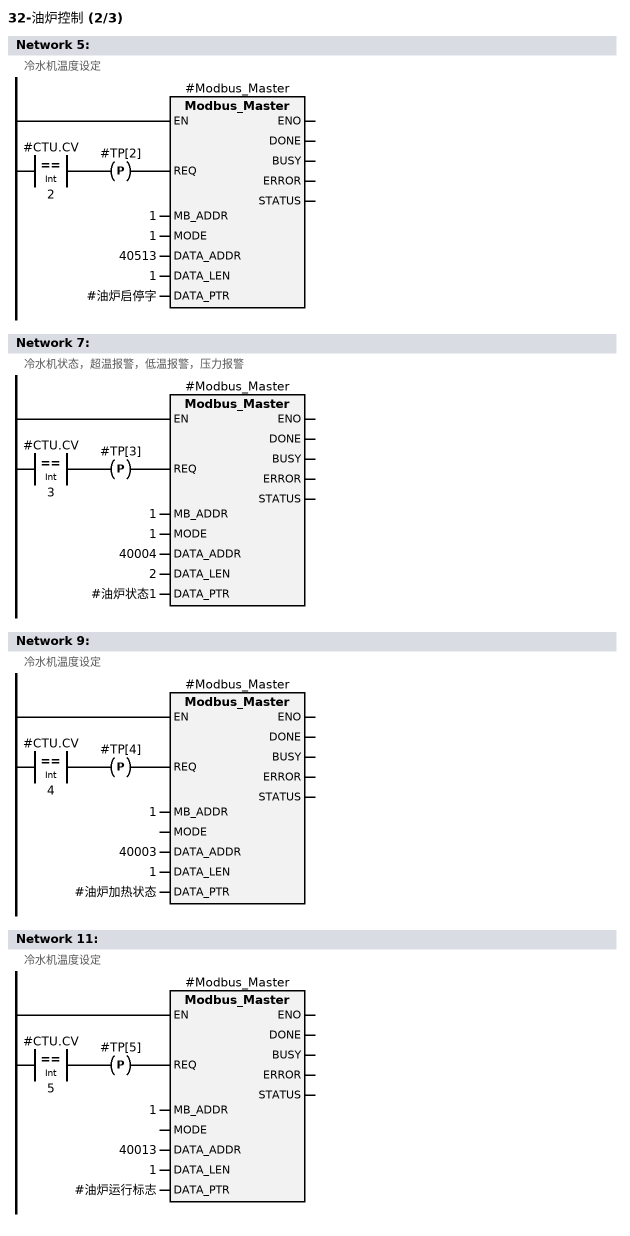
   RUNG wire#powerrail
      #Modbus_Master.Modbus_Master(REQ := wire#w1, MB_ADDR := 1, MODE := 1, DATA_ADDR := 40513, DATA_LEN := 1, DATA_PTR := #油炉启停字, DONE =>, BUSY =>, ERROR =>, STATUS =>)
   END_RUNG
   RUNG wire#powerrail
      { S7_Templates := "SrcType := Int" } EQ_Contact(in1 := #CTU.CV, in2 := 2)
      P_Trig( #TP[2] )
   END_RUNG wire#w1
   // the same network as SCL:
   #_w1 := #CTU.CV = 2;
   #_w2 := #_w1 AND NOT #TP[2];   // rising edge
   #TP[2] := #_w1;
   #Modbus_Master(REQ := #_w2, MB_ADDR := 1, MODE := 1, DATA_ADDR := 40513, DATA_LEN := 1, DATA_PTR := #油炉启停字);   // Modbus_Master
END_REGION

REGION Network 6 (SCL)
   IF #油炉循环泵启停 = TRUE THEN
       #油炉启停字:= 114;
   ELSE
       #油炉启停字 := 112;
   END_IF;
END_REGION

REGION Network 7
   // 冷水机状态，超温报警，低温报警，压力报警
   RUNG wire#powerrail
      #Modbus_Master.Modbus_Master(REQ := wire#w1, MB_ADDR := 1, MODE := 1, DATA_ADDR := 40004, DATA_LEN := 2, DATA_PTR := #油炉状态1, DONE =>, BUSY =>, ERROR =>, STATUS =>)
   END_RUNG
   RUNG wire#powerrail
      { S7_Templates := "SrcType := Int" } EQ_Contact(in1 := #CTU.CV, in2 := 3)
      P_Trig( #TP[3] )
   END_RUNG wire#w1
   // the same network as SCL:
   #_w1 := #CTU.CV = 3;
   #_w2 := #_w1 AND NOT #TP[3];   // rising edge
   #TP[3] := #_w1;
   #Modbus_Master(REQ := #_w2, MB_ADDR := 1, MODE := 1, DATA_ADDR := 40004, DATA_LEN := 2, DATA_PTR := #油炉状态1);   // Modbus_Master
END_REGION

REGION Network 8 (SCL)
   IF #油炉状态1>1 OR #油炉状态2>1 THEN
       #油炉报警 := TRUE;
   ELSE
       #油炉报警 := FALSE;
   END_IF;
END_REGION

REGION Network 9
   // 冷水机温度设定
   RUNG wire#powerrail
      #Modbus_Master.Modbus_Master(REQ := wire#w1, MB_ADDR := 1, MODE :=, DATA_ADDR := 40003, DATA_LEN := 1, DATA_PTR := #油炉加热状态, DONE =>, BUSY =>, ERROR =>, STATUS =>)
   END_RUNG
   RUNG wire#powerrail
      { S7_Templates := "SrcType := Int" } EQ_Contact(in1 := #CTU.CV, in2 := 4)
      P_Trig( #TP[4] )
   END_RUNG wire#w1
   // the same network as SCL:
   #_w1 := #CTU.CV = 4;
   #_w2 := #_w1 AND NOT #TP[4];   // rising edge
   #TP[4] := #_w1;
   #Modbus_Master(REQ := #_w2, MB_ADDR := 1, DATA_ADDR := 40003, DATA_LEN := 1, DATA_PTR := #油炉加热状态);   // Modbus_Master
END_REGION

REGION Network 10 (SCL)
   IF #油炉加热状态 >= 8 THEN
       #油炉冷却阀启停状态 := TRUE;
   ELSE
       #油炉冷却阀启停状态 := FALSE;
   END_IF;

   IF #油炉加热状态 >= 4 THEN
       #油炉加热泵启停状态 := TRUE;
   ELSE
       #油炉加热泵启停状态 := FALSE;
   END_IF;


   IF #油炉加热状态 >= 2 THEN
       #油炉加热器2状态 := TRUE;
   ELSE
       #油炉加热器2状态 := FALSE;
   END_IF;

   IF #油炉加热状态 >= 1 THEN
       #油炉加热器1状态 := TRUE;
   ELSE
       #油炉加热器1状态 := FALSE;
   END_IF;
END_REGION

REGION Network 11
   // 冷水机温度设定
   RUNG wire#powerrail
      #Modbus_Master.Modbus_Master(REQ := wire#w1, MB_ADDR := 1, MODE :=, DATA_ADDR := 40013, DATA_LEN := 1, DATA_PTR := #油炉运行标志, DONE =>, BUSY =>, ERROR =>, STATUS =>)
   END_RUNG
   RUNG wire#powerrail
      { S7_Templates := "SrcType := Int" } EQ_Contact(in1 := #CTU.CV, in2 := 5)
      P_Trig( #TP[5] )
   END_RUNG wire#w1
   // the same network as SCL:
   #_w1 := #CTU.CV = 5;
   #_w2 := #_w1 AND NOT #TP[5];   // rising edge
   #TP[5] := #_w1;
   #Modbus_Master(REQ := #_w2, MB_ADDR := 1, DATA_ADDR := 40013, DATA_LEN := 1, DATA_PTR := #油炉运行标志);   // Modbus_Master
END_REGION

REGION Network 12
   // 冷水机温du
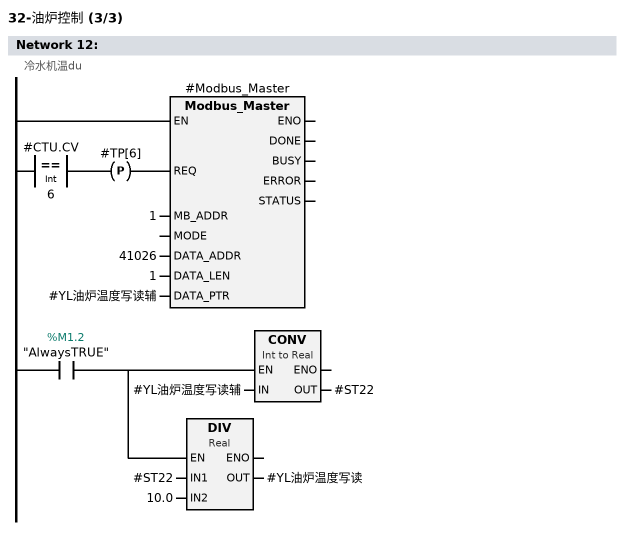
   RUNG wire#powerrail
      #Modbus_Master.Modbus_Master(REQ := wire#w1, MB_ADDR := 1, MODE :=, DATA_ADDR := 41026, DATA_LEN := 1, DATA_PTR := #YL油炉温度写读辅, DONE =>, BUSY =>, ERROR =>, STATUS =>)
   END_RUNG
   RUNG wire#powerrail
      { S7_Templates := "SrcType := Int" } EQ_Contact(in1 := #CTU.CV, in2 := 6)
      P_Trig( #TP[6] )
   END_RUNG wire#w1
   RUNG wire#powerrail
      Contact( "AlwaysTRUE" )
      wire#w2
      { S7_Templates := "[SrcType := Int, DestType := Real]" } Convert(in := #YL油炉温度写读辅, out => #ST22)
   END_RUNG
   RUNG wire#w2
      { S7_Templates := "SrcType := Real" } Div(in1 := #ST22, in2 := 10.0, out => #YL油炉温度写读)
   END_RUNG
   // the same network as SCL:
   #_w1 := #CTU.CV = 6;
   #_w2 := #_w1 AND NOT #TP[6];   // rising edge
   #TP[6] := #_w1;
   #Modbus_Master(REQ := #_w2, MB_ADDR := 1, DATA_ADDR := 41026, DATA_LEN := 1, DATA_PTR := #YL油炉温度写读辅);   // Modbus_Master
   IF "AlwaysTRUE" THEN
       #ST22 := INT_TO_REAL(#YL油炉温度写读辅);
       #YL油炉温度写读 := #ST22 / 10.0;
   END_IF;
END_REGION

REGION Network 13 (SCL)
   IF #油炉运行标志 >= 4 THEN
       #油炉强制冷却状态 := TRUE;
   ELSE
       #油炉强制冷却状态 := FALSE;
   END_IF;

   IF #油炉运行标志 >= 2 THEN
       #油炉自整定状态 := TRUE;
   ELSE
       #油炉自整定状态 := FALSE;
   END_IF;


   IF #油炉运行标志 >= 1 THEN
       #油炉运行状态 := TRUE;
   ELSE
       #油炉运行状态 := FALSE;
   END_IF;
END_REGION
END_FUNCTION_BLOCK

FUNCTION_BLOCK "33冷水机控制"   // FB5, LAD
{ S7_Optimized_Access := 'FALSE' }
VERSION : 0.1
// stored: AutoNumber true, IsIECCheckEnabled false, SetENOAutomatically false, UDAEnableTagReadback false
   VAR_IN_OUT
      冷水温度写 : Real;
      LS冷水温度写读 : Real;
      冷水温度读 : Real;
      冷水启停开关 : Bool;
      冷水报警 : Bool;
      机组状态 : Int;
   END_VAR
   VAR DB_SPECIFIC
      CTU { S7_SetPoint := 'True'} : CTU_INT;
      TEMP { S7_SetPoint := 'True'} : Bool;
      TP : Array[0..40] of Bool;
      冷水温度读辅 : Int;
      冷水温度写辅 : Int;
      LS冷水温度写读辅 : Int;
      ST1 : Real;
      ST2 : Real;
      ST3 : Real;
      ST4 : Real;
      ST5 : Real;
      ST16 : Real;
      ST17 : Real;
      ST18 : Real;
      ST20 : Real;
      ST21 : Real;
      ST22 : Real;
      ST23 : Array[0..2] of Int;
      冷水温度启停 : Int;
   END_VAR
   VAR
      Modbus_Comm_Load { S7_SetPoint := 'True'} : Modbus_Comm_Load;
      Modbus_Master { S7_SetPoint := 'True'} : Modbus_Master;
   END_VAR
   VAR_TEMP   // added for the SCL form of the ladder/FBD networks
      _w1 : Bool;
      _w2 : Bool;
      _w3 : Bool;
   END_VAR
BEGIN

REGION Network 1
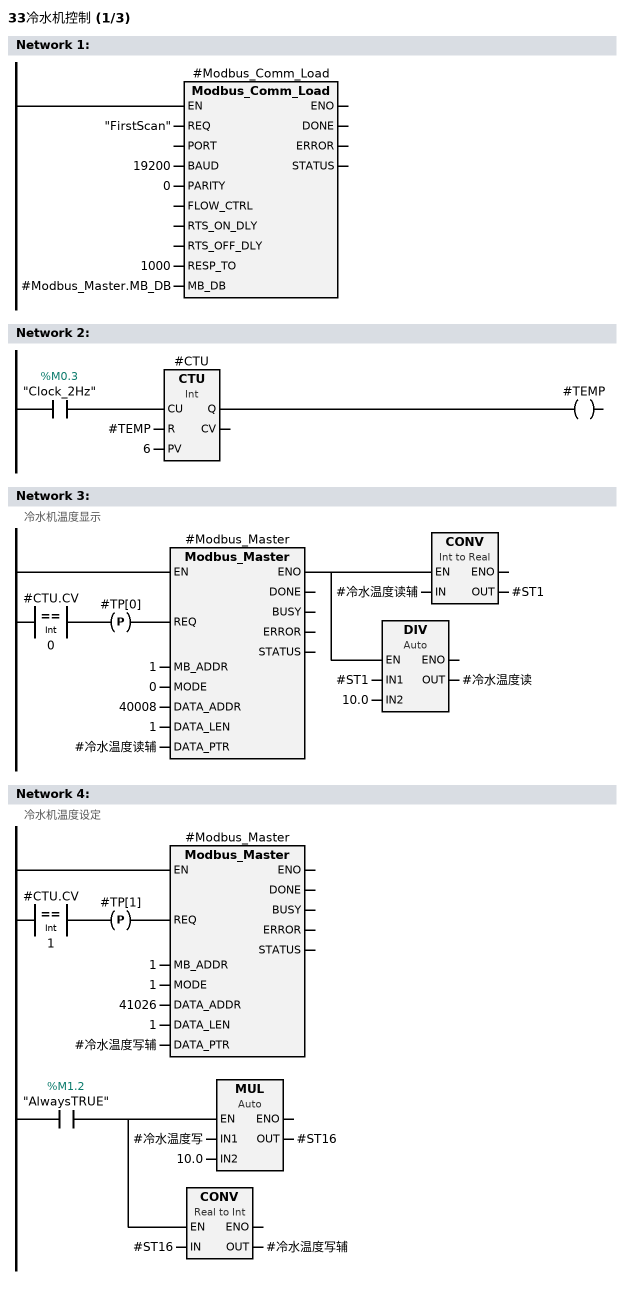
   RUNG wire#powerrail
      #Modbus_Comm_Load.Modbus_Comm_Load(REQ := "FirstScan", PORT :=, BAUD := 19200, PARITY := 0, FLOW_CTRL :=, RTS_ON_DLY :=, RTS_OFF_DLY :=, RESP_TO := 1000, MB_DB := #Modbus_Master.MB_DB, DONE =>, ERROR =>, STATUS =>)
   END_RUNG
   // the same network as SCL:
   #Modbus_Comm_Load(REQ := "FirstScan",   // Modbus_Comm_Load
                     BAUD := 19200,
                     PARITY := 0,
                     RESP_TO := 1000,
                     MB_DB := #Modbus_Master.MB_DB);
END_REGION

REGION Network 2
   RUNG wire#powerrail
      Contact( "Clock_2Hz" )
      { S7_Templates := "value_type := Int" } #CTU.CTU(r := #TEMP, pv := 6, cv =>)
      Coil( #TEMP )
   END_RUNG
   // the same network as SCL:
   #CTU(CU := "Clock_2Hz", R := #TEMP, PV := 6);   // CTU
   #TEMP := #CTU.Q;
END_REGION

REGION Network 3
   // 冷水机温度显示
   RUNG wire#powerrail
      #Modbus_Master.Modbus_Master(REQ := wire#w1, MB_ADDR := 1, MODE := 0, DATA_ADDR := 40008, DATA_LEN := 1, DATA_PTR := #冷水温度读辅, DONE =>, BUSY =>, ERROR =>, STATUS =>)
      wire#w2
      { S7_Templates := "[SrcType := Int, DestType := Real]" } Convert(in := #冷水温度读辅, out => #ST1)
   END_RUNG
   RUNG wire#powerrail
      { S7_Templates := "SrcType := Int" } EQ_Contact(in1 := #CTU.CV, in2 := 0)
      P_Trig( #TP[0] )
   END_RUNG wire#w1
   RUNG wire#w2
      Div(in1 := #ST1, in2 := 10.0, out => #冷水温度读)
   END_RUNG
   // the same network as SCL:
   #_w1 := #CTU.CV = 0;
   #_w2 := #_w1 AND NOT #TP[0];   // rising edge
   #TP[0] := #_w1;
   #Modbus_Master(REQ := #_w2,   // Modbus_Master
                  MB_ADDR := 1,
                  MODE := 0,
                  DATA_ADDR := 40008,
                  DATA_LEN := 1,
                  DATA_PTR := #冷水温度读辅,
                  ENO => #_w3);
   IF #_w3 THEN
       #ST1 := INT_TO_REAL(#冷水温度读辅);
       #冷水温度读 := #ST1 / 10.0;
   END_IF;
END_REGION

REGION Network 4
   // 冷水机温度设定
   RUNG wire#powerrail
      #Modbus_Master.Modbus_Master(REQ := wire#w1, MB_ADDR := 1, MODE := 1, DATA_ADDR := 41026, DATA_LEN := 1, DATA_PTR := #冷水温度写辅, DONE =>, BUSY =>, ERROR =>, STATUS =>)
   END_RUNG
   RUNG wire#powerrail
      { S7_Templates := "SrcType := Int" } EQ_Contact(in1 := #CTU.CV, in2 := 1)
      P_Trig( #TP[1] )
   END_RUNG wire#w1
   RUNG wire#powerrail
      Contact( "AlwaysTRUE" )
      wire#w2
      Mul(in1 := #冷水温度写, in2 := 10.0, out => #ST16)
   END_RUNG
   RUNG wire#w2
      { S7_Templates := "[SrcType := Real, DestType := Int]" } Convert(in := #ST16, out => #冷水温度写辅)
   END_RUNG
   // the same network as SCL:
   #_w1 := #CTU.CV = 1;
   #_w2 := #_w1 AND NOT #TP[1];   // rising edge
   #TP[1] := #_w1;
   #Modbus_Master(REQ := #_w2, MB_ADDR := 1, MODE := 1, DATA_ADDR := 41026, DATA_LEN := 1, DATA_PTR := #冷水温度写辅);   // Modbus_Master
   IF "AlwaysTRUE" THEN
       #ST16 := #冷水温度写 * 10.0;
       #冷水温度写辅 := REAL_TO_INT(#ST16);
   END_IF;
END_REGION

REGION Network 5
   // 冷水机启停，11100，关，11110开
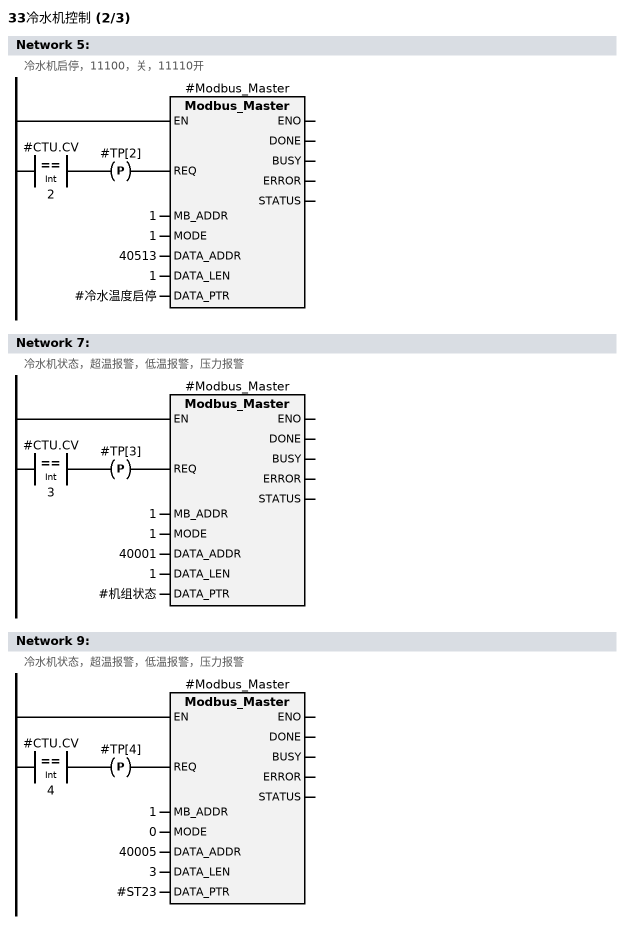
   RUNG wire#powerrail
      #Modbus_Master.Modbus_Master(REQ := wire#w1, MB_ADDR := 1, MODE := 1, DATA_ADDR := 40513, DATA_LEN := 1, DATA_PTR := #冷水温度启停, DONE =>, BUSY =>, ERROR =>, STATUS =>)
   END_RUNG
   RUNG wire#powerrail
      { S7_Templates := "SrcType := Int" } EQ_Contact(in1 := #CTU.CV, in2 := 2)
      P_Trig( #TP[2] )
   END_RUNG wire#w1
   // the same network as SCL:
   #_w1 := #CTU.CV = 2;
   #_w2 := #_w1 AND NOT #TP[2];   // rising edge
   #TP[2] := #_w1;
   #Modbus_Master(REQ := #_w2, MB_ADDR := 1, MODE := 1, DATA_ADDR := 40513, DATA_LEN := 1, DATA_PTR := #冷水温度启停);   // Modbus_Master
END_REGION

REGION Network 6 (SCL)
   IF #冷水启停开关 = TRUE THEN
       #冷水温度启停 := 114;

   END_IF;

   IF #冷水启停开关 = FALSE THEN
       #冷水温度启停 := 112;

   END_IF;
END_REGION

REGION Network 7
   // 冷水机状态，超温报警，低温报警，压力报警
   RUNG wire#powerrail
      #Modbus_Master.Modbus_Master(REQ := wire#w1, MB_ADDR := 1, MODE := 1, DATA_ADDR := 40001, DATA_LEN := 1, DATA_PTR := #机组状态, DONE =>, BUSY =>, ERROR =>, STATUS =>)
   END_RUNG
   RUNG wire#powerrail
      { S7_Templates := "SrcType := Int" } EQ_Contact(in1 := #CTU.CV, in2 := 3)
      P_Trig( #TP[3] )
   END_RUNG wire#w1
   // the same network as SCL:
   #_w1 := #CTU.CV = 3;
   #_w2 := #_w1 AND NOT #TP[3];   // rising edge
   #TP[3] := #_w1;
   #Modbus_Master(REQ := #_w2, MB_ADDR := 1, MODE := 1, DATA_ADDR := 40001, DATA_LEN := 1, DATA_PTR := #机组状态);   // Modbus_Master
END_REGION

REGION Network 9
   // 冷水机状态，超温报警，低温报警，压力报警
   RUNG wire#powerrail
      #Modbus_Master.Modbus_Master(REQ := wire#w1, MB_ADDR := 1, MODE := 0, DATA_ADDR := 40005, DATA_LEN := 3, DATA_PTR := #ST23, DONE =>, BUSY =>, ERROR =>, STATUS =>)
   END_RUNG
   RUNG wire#powerrail
      { S7_Templates := "SrcType := Int" } EQ_Contact(in1 := #CTU.CV, in2 := 4)
      P_Trig( #TP[4] )
   END_RUNG wire#w1
   // the same network as SCL:
   #_w1 := #CTU.CV = 4;
   #_w2 := #_w1 AND NOT #TP[4];   // rising edge
   #TP[4] := #_w1;
   #Modbus_Master(REQ := #_w2, MB_ADDR := 1, MODE := 0, DATA_ADDR := 40005, DATA_LEN := 3, DATA_PTR := #ST23);   // Modbus_Master
END_REGION

REGION Network 10 (SCL)
   IF #ST23[0]>0 OR #ST23[1]>0 OR #ST23[2]>0 THEN
       #冷水报警 := 1;
   ELSE
       #冷水报警 :=0;
   END_IF;
END_REGION

REGION Network 11
   // 冷水机温du
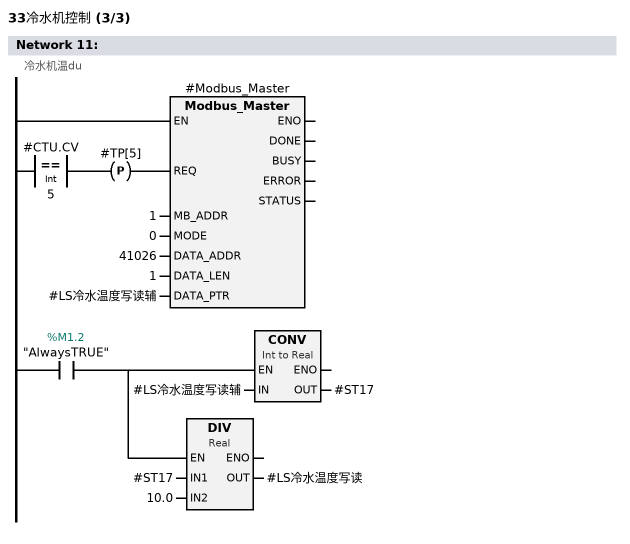
   RUNG wire#powerrail
      #Modbus_Master.Modbus_Master(REQ := wire#w1, MB_ADDR := 1, MODE := 0, DATA_ADDR := 41026, DATA_LEN := 1, DATA_PTR := #LS冷水温度写读辅, DONE =>, BUSY =>, ERROR =>, STATUS =>)
   END_RUNG
   RUNG wire#powerrail
      { S7_Templates := "SrcType := Int" } EQ_Contact(in1 := #CTU.CV, in2 := 5)
      P_Trig( #TP[5] )
   END_RUNG wire#w1
   RUNG wire#powerrail
      Contact( "AlwaysTRUE" )
      wire#w2
      { S7_Templates := "[SrcType := Int, DestType := Real]" } Convert(in := #LS冷水温度写读辅, out => #ST17)
   END_RUNG
   RUNG wire#w2
      { S7_Templates := "SrcType := Real" } Div(in1 := #ST17, in2 := 10.0, out => #LS冷水温度写读)
   END_RUNG
   // the same network as SCL:
   #_w1 := #CTU.CV = 5;
   #_w2 := #_w1 AND NOT #TP[5];   // rising edge
   #TP[5] := #_w1;
   #Modbus_Master(REQ := #_w2,   // Modbus_Master
                  MB_ADDR := 1,
                  MODE := 0,
                  DATA_ADDR := 41026,
                  DATA_LEN := 1,
                  DATA_PTR := #LS冷水温度写读辅);
   IF "AlwaysTRUE" THEN
       #ST17 := INT_TO_REAL(#LS冷水温度写读辅);
       #LS冷水温度写读 := #ST17 / 10.0;
   END_IF;
END_REGION
END_FUNCTION_BLOCK

FUNCTION_BLOCK "34仪表控制"   // FB45, LAD
{ S7_Optimized_Access := 'FALSE' }
VERSION : 0.1
// stored: AutoNumber true, IsIECCheckEnabled false, SetENOAutomatically false, UDAEnableTagReadback false
   VAR_OUTPUT
      动态 : Bool;
      稳态 : Bool;
      非零位 : Bool;
      零位 : Bool;
      毛重模式 : Bool;
      净重模式 : Bool;
      没有上超载 : Bool;
      上超载 : Bool;
      没有下超载 : Bool;
      下超载 : Bool;
      低位量程内 : Bool;
      高位量程内 : Bool;
      正常显示重量 : Bool;
      分度值缩小10倍显示重量 : Bool;
      A瞬时流量 : Real;
      A瞬时流量AT AT A瞬时流量 : Array[0..1] of Word;
      A瞬时流速 : Real;
      A瞬时流速AT AT A瞬时流速 : Array[0..1] of Word;
      A当前电流 : Real;
      A当前电流AT AT A当前电流 : Array[0..1] of Word;
      A介质温度 : Real;
      A介质温度AT AT A介质温度 : Array[0..1] of Word;
      A当前采集 : Real;
      A当前采集AT AT A当前采集 : Array[0..1] of Word;
      A流速下限 : Real;
      A流速下限AT AT A流速下限 : Array[0..1] of Word;
      A流速上限 : Real;
      A流速上限AT AT A流速上限 : Array[0..1] of Word;
      A管道内径 : Real;
      A管道内径AT AT A管道内径 : Array[0..1] of Word;
      B瞬时流量 : Real;
      B瞬时流量AT AT B瞬时流量 : Array[0..1] of Word;
      B瞬时流速 : Real;
      B瞬时流速AT AT B瞬时流速 : Array[0..1] of Word;
      B当前电流 : Real;
      B当前电流AT AT B当前电流 : Array[0..1] of Word;
      B介质温度 : Real;
      B介质温度AT AT B介质温度 : Array[0..1] of Word;
      B当前采集 : Real;
      B当前采集AT AT B当前采集 : Array[0..1] of Word;
      B流速下限 : Real;
      B流速下限AT AT B流速下限 : Array[0..1] of Word;
      B流速上限 : Real;
      B流速上限AT AT B流速上限 : Array[0..1] of Word;
      B管道内径 : Real;
      B管道内径AT AT B管道内径 : Array[0..1] of Word;
   END_VAR
   VAR_IN_OUT
      "秤操作-清零" : Bool;
      "秤操作-去皮" : Bool;
      "秤操作-清皮" : Bool;
      读重量 : Real;
   END_VAR
   VAR DB_SPECIFIC
      CTU { S7_SetPoint := 'True'} : CTU_INT;
      TEMP { S7_SetPoint := 'True'} : Bool;
      TON1 : TON_TIME;
      TP : Array[0..40] of Bool;
      秤操作辅助 : Int;
      CZTFZ : Int;
   END_VAR
   VAR
      CZT AT CZTFZ : Array[0..15] of Bool;
   END_VAR
   VAR DB_SPECIFIC
      ST1 : Array[0..5] of Word;
      ST2 : Array[0..7] of Word;
      ST3 : Array[0..1] of Word;
      ST4 : Array[0..5] of Word;
      ST5 : Array[0..7] of Word;
      ST6 : Array[0..1] of Word;
      ST7 : Array[0..1] of Word;
      读重量辅助 : DInt;
   END_VAR
   VAR
      读重量辅助AT AT 读重量辅助 : Array[0..1] of Word;
      Modbus_Comm_Load { S7_SetPoint := 'True'} : Modbus_Comm_Load;
      Modbus_Master { S7_SetPoint := 'True'} : Modbus_Master;
   END_VAR
   VAR_TEMP   // added for the SCL form of the ladder/FBD networks
      _w1 : Bool;
      _w2 : Bool;
      _w3 : Bool;
   END_VAR
BEGIN

REGION Network 1
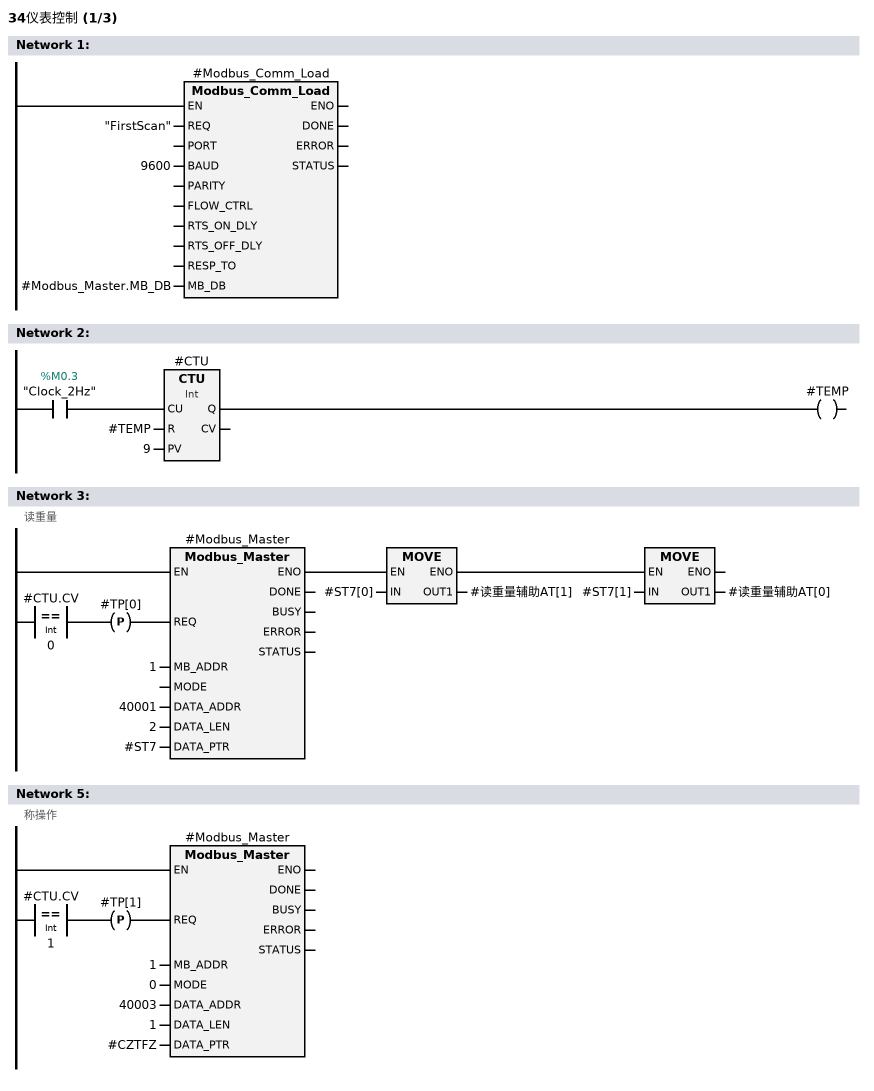
   RUNG wire#powerrail
      #Modbus_Comm_Load.Modbus_Comm_Load(REQ := "FirstScan", PORT :=, BAUD := 9600, PARITY :=, FLOW_CTRL :=, RTS_ON_DLY :=, RTS_OFF_DLY :=, RESP_TO :=, MB_DB := #Modbus_Master.MB_DB, DONE =>, ERROR =>, STATUS =>)
   END_RUNG
   // the same network as SCL:
   #Modbus_Comm_Load(REQ := "FirstScan", BAUD := 9600, MB_DB := #Modbus_Master.MB_DB);   // Modbus_Comm_Load
END_REGION

REGION Network 2
   RUNG wire#powerrail
      Contact( "Clock_2Hz" )
      { S7_Templates := "value_type := Int" } #CTU.CTU(r := #TEMP, pv := 9, cv =>)
      Coil( #TEMP )
   END_RUNG
   // the same network as SCL:
   #CTU(CU := "Clock_2Hz", R := #TEMP, PV := 9);   // CTU
   #TEMP := #CTU.Q;
END_REGION

REGION Network 3
   // 读重量
   RUNG wire#powerrail
      #Modbus_Master.Modbus_Master(REQ := wire#w1, MB_ADDR := 1, MODE :=, DATA_ADDR := 40001, DATA_LEN := 2, DATA_PTR := #ST7, DONE =>, BUSY =>, ERROR =>, STATUS =>)
      Move(in := #ST7[0], out1 => #读重量辅助AT[1])
      Move(in := #ST7[1], out1 => #读重量辅助AT[0])
   END_RUNG
   RUNG wire#powerrail
      { S7_Templates := "SrcType := Int" } EQ_Contact(in1 := #CTU.CV, in2 := 0)
      P_Trig( #TP[0] )
   END_RUNG wire#w1
   // the same network as SCL:
   #_w1 := #CTU.CV = 0;
   #_w2 := #_w1 AND NOT #TP[0];   // rising edge
   #TP[0] := #_w1;
   #Modbus_Master(REQ := #_w2, MB_ADDR := 1, DATA_ADDR := 40001, DATA_LEN := 2, DATA_PTR := #ST7, ENO => #_w3);   // Modbus_Master
   IF #_w3 THEN
       #读重量辅助AT[1] := #ST7[0];
       #读重量辅助AT[0] := #ST7[1];
   END_IF;
END_REGION

REGION Network 4 (SCL)


   #读重量 := DINT_TO_REAL(#读重量辅助) * 0.01;
END_REGION

REGION Network 5
   // 称操作
   RUNG wire#powerrail
      #Modbus_Master.Modbus_Master(REQ := wire#w1, MB_ADDR := 1, MODE := 0, DATA_ADDR := 40003, DATA_LEN := 1, DATA_PTR := #CZTFZ, DONE =>, BUSY =>, ERROR =>, STATUS =>)
   END_RUNG
   RUNG wire#powerrail
      { S7_Templates := "SrcType := Int" } EQ_Contact(in1 := #CTU.CV, in2 := 1)
      P_Trig( #TP[1] )
   END_RUNG wire#w1
   // the same network as SCL:
   #_w1 := #CTU.CV = 1;
   #_w2 := #_w1 AND NOT #TP[1];   // rising edge
   #TP[1] := #_w1;
   #Modbus_Master(REQ := #_w2, MB_ADDR := 1, MODE := 0, DATA_ADDR := 40003, DATA_LEN := 1, DATA_PTR := #CZTFZ);   // Modbus_Master
END_REGION

REGION Network 6 (SCL)
   IF #CZT[0] = TRUE THEN
       #动态 := 1;
       #稳态 := 0;
   ELSE
       #动态 := 0;
       #稳态 := 1;
   END_IF;

   IF #CZT[1] = TRUE THEN
       #非零位 := 1;
       #零位 := 0;
   ELSE
       #非零位 := 0;
       #零位 := 1;
   END_IF;


   IF #CZT[2] = TRUE THEN
       #毛重模式 := 1;
       #净重模式 := 0;
   ELSE
       #毛重模式 := 0;
       #净重模式 := 1;
   END_IF;


   IF #CZT[3] = TRUE THEN
       #没有上超载 := 1;
       #上超载 := 0;
   ELSE
       #没有上超载 := 0;
       #上超载 := 1;
   END_IF;


   IF #CZT[4] = TRUE THEN
       #没有下超载 := 1;
       #下超载 := 0;
   ELSE
       #没有下超载 := 0;
       #下超载 := 1;
   END_IF;


   IF #CZT[5] = TRUE THEN
       #低位量程内 := 1;
       #高位量程内 := 0;
   ELSE
       #低位量程内 := 0;
       #高位量程内 := 1;
   END_IF;


   IF #CZT[6] = TRUE THEN
       #正常显示重量 := 1;
       #分度值缩小10倍显示重量 := 0;
   ELSE
       #正常显示重量 := 0;
       #分度值缩小10倍显示重量 := 1;
   END_IF;
END_REGION

REGION Network 7
   // 称操作
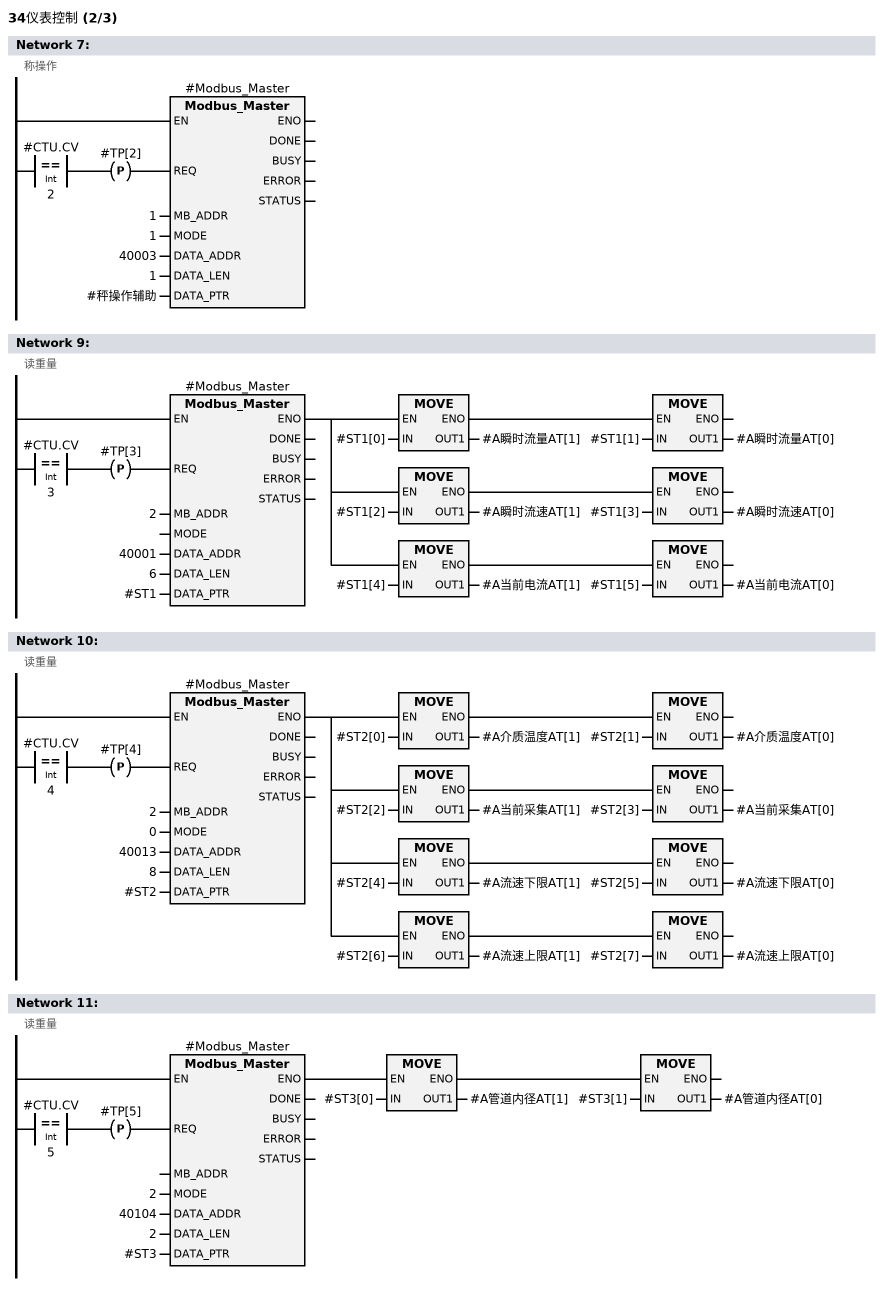
   RUNG wire#powerrail
      #Modbus_Master.Modbus_Master(REQ := wire#w1, MB_ADDR := 1, MODE := 1, DATA_ADDR := 40003, DATA_LEN := 1, DATA_PTR := #秤操作辅助, DONE =>, BUSY =>, ERROR =>, STATUS =>)
   END_RUNG
   RUNG wire#powerrail
      { S7_Templates := "SrcType := Int" } EQ_Contact(in1 := #CTU.CV, in2 := 2)
      P_Trig( #TP[2] )
   END_RUNG wire#w1
   // the same network as SCL:
   #_w1 := #CTU.CV = 2;
   #_w2 := #_w1 AND NOT #TP[2];   // rising edge
   #TP[2] := #_w1;
   #Modbus_Master(REQ := #_w2, MB_ADDR := 1, MODE := 1, DATA_ADDR := 40003, DATA_LEN := 1, DATA_PTR := #秤操作辅助);   // Modbus_Master
END_REGION

REGION Network 8 (SCL)
   IF #"秤操作-清零" = TRUE THEN
       #秤操作辅助 := 1;
       #"秤操作-清零" := 0;
   END_IF;

   IF #"秤操作-去皮" = TRUE THEN
       #秤操作辅助 := 2;
       #"秤操作-去皮" := 0;

   END_IF;
   IF #"秤操作-清皮" = TRUE THEN
       #秤操作辅助 := 3;
       #"秤操作-清皮" := 0;

   END_IF;


   #TON1(IN := #秤操作辅助<>0,
         PT := T#5S);

   IF #TON1.Q THEN
       #秤操作辅助 := 0;

   END_IF;
END_REGION

REGION Network 9
   // 读重量
   RUNG wire#powerrail
      #Modbus_Master.Modbus_Master(REQ := wire#w1, MB_ADDR := 2, MODE :=, DATA_ADDR := 40001, DATA_LEN := 6, DATA_PTR := #ST1, DONE =>, BUSY =>, ERROR =>, STATUS =>)
      wire#w2
      Move(in := #ST1[0], out1 => #A瞬时流量AT[1])
      Move(in := #ST1[1], out1 => #A瞬时流量AT[0])
   END_RUNG
   RUNG wire#powerrail
      { S7_Templates := "SrcType := Int" } EQ_Contact(in1 := #CTU.CV, in2 := 3)
      P_Trig( #TP[3] )
   END_RUNG wire#w1
   RUNG wire#w2
      Move(in := #ST1[2], out1 => #A瞬时流速AT[1])
      Move(in := #ST1[3], out1 => #A瞬时流速AT[0])
   END_RUNG
   RUNG wire#w2
      Move(in := #ST1[4], out1 => #A当前电流AT[1])
      Move(in := #ST1[5], out1 => #A当前电流AT[0])
   END_RUNG
   // the same network as SCL:
   #_w1 := #CTU.CV = 3;
   #_w2 := #_w1 AND NOT #TP[3];   // rising edge
   #TP[3] := #_w1;
   #Modbus_Master(REQ := #_w2, MB_ADDR := 2, DATA_ADDR := 40001, DATA_LEN := 6, DATA_PTR := #ST1, ENO => #_w3);   // Modbus_Master
   IF #_w3 THEN
       #A瞬时流量AT[1] := #ST1[0];
       #A瞬时流量AT[0] := #ST1[1];
       #A瞬时流速AT[1] := #ST1[2];
       #A瞬时流速AT[0] := #ST1[3];
       #A当前电流AT[1] := #ST1[4];
       #A当前电流AT[0] := #ST1[5];
   END_IF;
END_REGION

REGION Network 10
   // 读重量
   RUNG wire#powerrail
      #Modbus_Master.Modbus_Master(REQ := wire#w1, MB_ADDR := 2, MODE := 0, DATA_ADDR := 40013, DATA_LEN := 8, DATA_PTR := #ST2, DONE =>, BUSY =>, ERROR =>, STATUS =>)
      wire#w2
      Move(in := #ST2[0], out1 => #A介质温度AT[1])
      Move(in := #ST2[1], out1 => #A介质温度AT[0])
   END_RUNG
   RUNG wire#powerrail
      { S7_Templates := "SrcType := Int" } EQ_Contact(in1 := #CTU.CV, in2 := 4)
      P_Trig( #TP[4] )
   END_RUNG wire#w1
   RUNG wire#w2
      Move(in := #ST2[2], out1 => #A当前采集AT[1])
      Move(in := #ST2[3], out1 => #A当前采集AT[0])
   END_RUNG
   RUNG wire#w2
      Move(in := #ST2[4], out1 => #A流速下限AT[1])
      Move(in := #ST2[5], out1 => #A流速下限AT[0])
   END_RUNG
   RUNG wire#w2
      Move(in := #ST2[6], out1 => #A流速上限AT[1])
      Move(in := #ST2[7], out1 => #A流速上限AT[0])
   END_RUNG
   // the same network as SCL:
   #_w1 := #CTU.CV = 4;
   #_w2 := #_w1 AND NOT #TP[4];   // rising edge
   #TP[4] := #_w1;
   #Modbus_Master(REQ := #_w2,   // Modbus_Master
                  MB_ADDR := 2,
                  MODE := 0,
                  DATA_ADDR := 40013,
                  DATA_LEN := 8,
                  DATA_PTR := #ST2,
                  ENO => #_w3);
   IF #_w3 THEN
       #A介质温度AT[1] := #ST2[0];
       #A介质温度AT[0] := #ST2[1];
       #A当前采集AT[1] := #ST2[2];
       #A当前采集AT[0] := #ST2[3];
       #A流速下限AT[1] := #ST2[4];
       #A流速下限AT[0] := #ST2[5];
       #A流速上限AT[1] := #ST2[6];
       #A流速上限AT[0] := #ST2[7];
   END_IF;
END_REGION

REGION Network 11
   // 读重量
   RUNG wire#powerrail
      #Modbus_Master.Modbus_Master(REQ := wire#w1, MB_ADDR :=, MODE := 2, DATA_ADDR := 40104, DATA_LEN := 2, DATA_PTR := #ST3, DONE =>, BUSY =>, ERROR =>, STATUS =>)
      Move(in := #ST3[0], out1 => #A管道内径AT[1])
      Move(in := #ST3[1], out1 => #A管道内径AT[0])
   END_RUNG
   RUNG wire#powerrail
      { S7_Templates := "SrcType := Int" } EQ_Contact(in1 := #CTU.CV, in2 := 5)
      P_Trig( #TP[5] )
   END_RUNG wire#w1
   // the same network as SCL:
   #_w1 := #CTU.CV = 5;
   #_w2 := #_w1 AND NOT #TP[5];   // rising edge
   #TP[5] := #_w1;
   #Modbus_Master(REQ := #_w2, MODE := 2, DATA_ADDR := 40104, DATA_LEN := 2, DATA_PTR := #ST3, ENO => #_w3);   // Modbus_Master
   IF #_w3 THEN
       #A管道内径AT[1] := #ST3[0];
       #A管道内径AT[0] := #ST3[1];
   END_IF;
END_REGION

REGION Network 12
   // 读重量
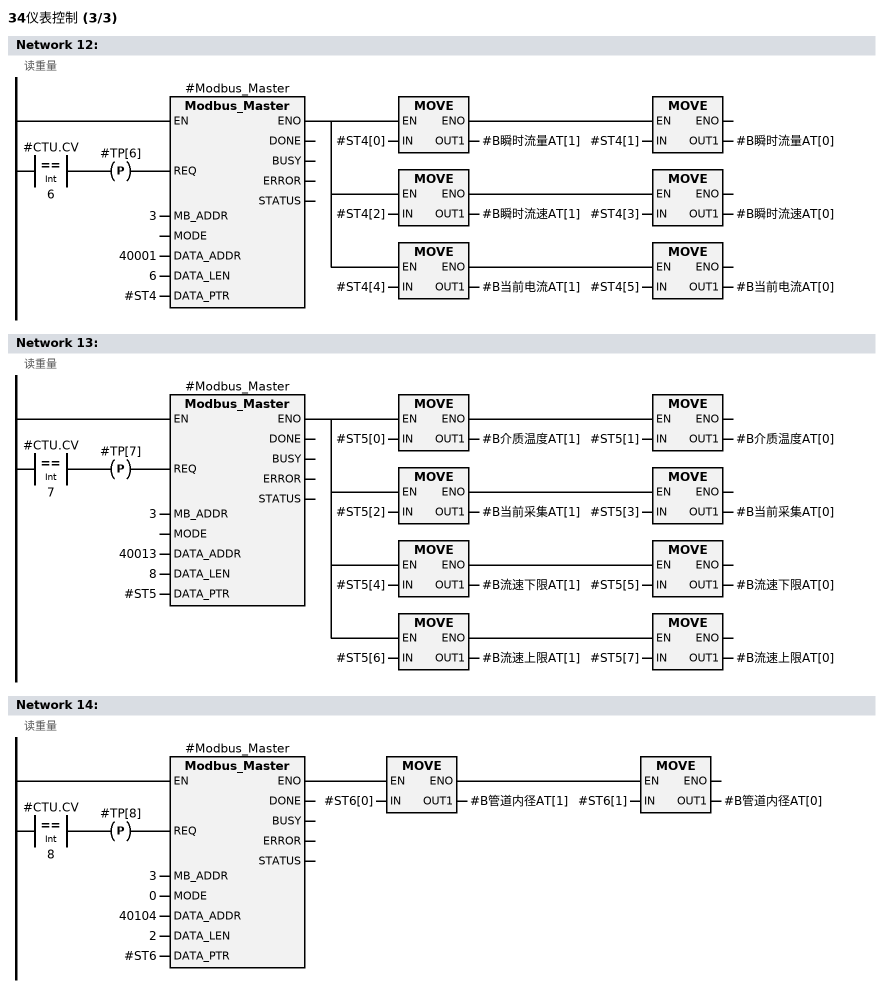
   RUNG wire#powerrail
      #Modbus_Master.Modbus_Master(REQ := wire#w1, MB_ADDR := 3, MODE :=, DATA_ADDR := 40001, DATA_LEN := 6, DATA_PTR := #ST4, DONE =>, BUSY =>, ERROR =>, STATUS =>)
      wire#w2
      Move(in := #ST4[0], out1 => #B瞬时流量AT[1])
      Move(in := #ST4[1], out1 => #B瞬时流量AT[0])
   END_RUNG
   RUNG wire#powerrail
      { S7_Templates := "SrcType := Int" } EQ_Contact(in1 := #CTU.CV, in2 := 6)
      P_Trig( #TP[6] )
   END_RUNG wire#w1
   RUNG wire#w2
      Move(in := #ST4[2], out1 => #B瞬时流速AT[1])
      Move(in := #ST4[3], out1 => #B瞬时流速AT[0])
   END_RUNG
   RUNG wire#w2
      Move(in := #ST4[4], out1 => #B当前电流AT[1])
      Move(in := #ST4[5], out1 => #B当前电流AT[0])
   END_RUNG
   // the same network as SCL:
   #_w1 := #CTU.CV = 6;
   #_w2 := #_w1 AND NOT #TP[6];   // rising edge
   #TP[6] := #_w1;
   #Modbus_Master(REQ := #_w2, MB_ADDR := 3, DATA_ADDR := 40001, DATA_LEN := 6, DATA_PTR := #ST4, ENO => #_w3);   // Modbus_Master
   IF #_w3 THEN
       #B瞬时流量AT[1] := #ST4[0];
       #B瞬时流量AT[0] := #ST4[1];
       #B瞬时流速AT[1] := #ST4[2];
       #B瞬时流速AT[0] := #ST4[3];
       #B当前电流AT[1] := #ST4[4];
       #B当前电流AT[0] := #ST4[5];
   END_IF;
END_REGION

REGION Network 13
   // 读重量
   RUNG wire#powerrail
      #Modbus_Master.Modbus_Master(REQ := wire#w1, MB_ADDR := 3, MODE :=, DATA_ADDR := 40013, DATA_LEN := 8, DATA_PTR := #ST5, DONE =>, BUSY =>, ERROR =>, STATUS =>)
      wire#w2
      Move(in := #ST5[0], out1 => #B介质温度AT[1])
      Move(in := #ST5[1], out1 => #B介质温度AT[0])
   END_RUNG
   RUNG wire#powerrail
      { S7_Templates := "SrcType := Int" } EQ_Contact(in1 := #CTU.CV, in2 := 7)
      P_Trig( #TP[7] )
   END_RUNG wire#w1
   RUNG wire#w2
      Move(in := #ST5[2], out1 => #B当前采集AT[1])
      Move(in := #ST5[3], out1 => #B当前采集AT[0])
   END_RUNG
   RUNG wire#w2
      Move(in := #ST5[4], out1 => #B流速下限AT[1])
      Move(in := #ST5[5], out1 => #B流速下限AT[0])
   END_RUNG
   RUNG wire#w2
      Move(in := #ST5[6], out1 => #B流速上限AT[1])
      Move(in := #ST5[7], out1 => #B流速上限AT[0])
   END_RUNG
   // the same network as SCL:
   #_w1 := #CTU.CV = 7;
   #_w2 := #_w1 AND NOT #TP[7];   // rising edge
   #TP[7] := #_w1;
   #Modbus_Master(REQ := #_w2, MB_ADDR := 3, DATA_ADDR := 40013, DATA_LEN := 8, DATA_PTR := #ST5, ENO => #_w3);   // Modbus_Master
   IF #_w3 THEN
       #B介质温度AT[1] := #ST5[0];
       #B介质温度AT[0] := #ST5[1];
       #B当前采集AT[1] := #ST5[2];
       #B当前采集AT[0] := #ST5[3];
       #B流速下限AT[1] := #ST5[4];
       #B流速下限AT[0] := #ST5[5];
       #B流速上限AT[1] := #ST5[6];
       #B流速上限AT[0] := #ST5[7];
   END_IF;
END_REGION

REGION Network 14
   // 读重量
   RUNG wire#powerrail
      #Modbus_Master.Modbus_Master(REQ := wire#w1, MB_ADDR := 3, MODE := 0, DATA_ADDR := 40104, DATA_LEN := 2, DATA_PTR := #ST6, DONE =>, BUSY =>, ERROR =>, STATUS =>)
      Move(in := #ST6[0], out1 => #B管道内径AT[1])
      Move(in := #ST6[1], out1 => #B管道内径AT[0])
   END_RUNG
   RUNG wire#powerrail
      { S7_Templates := "SrcType := Int" } EQ_Contact(in1 := #CTU.CV, in2 := 8)
      P_Trig( #TP[8] )
   END_RUNG wire#w1
   // the same network as SCL:
   #_w1 := #CTU.CV = 8;
   #_w2 := #_w1 AND NOT #TP[8];   // rising edge
   #TP[8] := #_w1;
   #Modbus_Master(REQ := #_w2,   // Modbus_Master
                  MB_ADDR := 3,
                  MODE := 0,
                  DATA_ADDR := 40104,
                  DATA_LEN := 2,
                  DATA_PTR := #ST6,
                  ENO => #_w3);
   IF #_w3 THEN
       #B管道内径AT[1] := #ST6[0];
       #B管道内径AT[0] := #ST6[1];
   END_IF;
END_REGION
END_FUNCTION_BLOCK

FUNCTION_BLOCK "冷水机控制"   // FB50, LAD
{ S7_Optimized_Access := 'FALSE' }
VERSION : 0.1
// stored: AutoNumber true, IsIECCheckEnabled false, SetENOAutomatically false, UDAEnableTagReadback false
   VAR_IN_OUT
      冷水温度写 : Real;
      LS冷水温度写读 : Real;
      冷水温度读 : Real;
      冷水启停开关 : Bool;
      冷水报警 : Bool;
      机组状态 : Int;
   END_VAR
   VAR DB_SPECIFIC
      CTU { S7_SetPoint := 'True'} : CTU_INT;
      TEMP { S7_SetPoint := 'True'} : Bool;
      TP : Array[0..40] of Bool;
      冷水温度读辅 : Int;
      冷水温度写辅 : Int;
      LS冷水温度写读辅 : Int;
      ST1 : Real;
      ST2 : Real;
      ST3 : Real;
      ST4 : Real;
      ST5 : Real;
      ST16 : Real;
      ST17 : Real;
      ST18 : Real;
      ST20 : Real;
      ST21 : Real;
      ST22 : Real;
      ST23 : Array[0..2] of Int;
      冷水温度启停 : Int;
   END_VAR
   VAR
      Modbus_Comm_Load_ { S7_SetPoint := 'True'} : Modbus_Comm_Load;
      Modbus_Master { S7_SetPoint := 'True'} : Modbus_Master;
   END_VAR
   VAR_TEMP   // added for the SCL form of the ladder/FBD networks
      _w1 : Bool;
      _w2 : Bool;
      _w3 : Bool;
   END_VAR
BEGIN

REGION Network 1
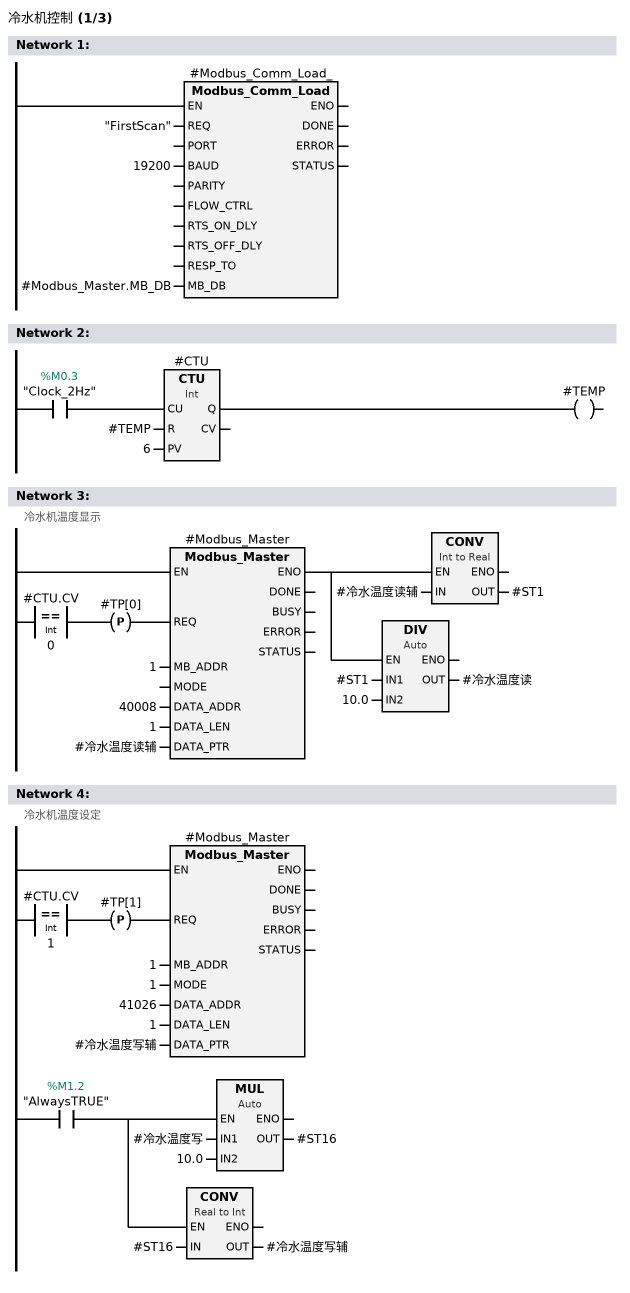
   RUNG wire#powerrail
      #Modbus_Comm_Load_.Modbus_Comm_Load(REQ := "FirstScan", PORT :=, BAUD := 19200, PARITY :=, FLOW_CTRL :=, RTS_ON_DLY :=, RTS_OFF_DLY :=, RESP_TO :=, MB_DB := #Modbus_Master.MB_DB, DONE =>, ERROR =>, STATUS =>)
   END_RUNG
   // the same network as SCL:
   #Modbus_Comm_Load_(REQ := "FirstScan", BAUD := 19200, MB_DB := #Modbus_Master.MB_DB);   // Modbus_Comm_Load
END_REGION

REGION Network 2
   RUNG wire#powerrail
      Contact( "Clock_2Hz" )
      { S7_Templates := "value_type := Int" } #CTU.CTU(r := #TEMP, pv := 6, cv =>)
      Coil( #TEMP )
   END_RUNG
   // the same network as SCL:
   #CTU(CU := "Clock_2Hz", R := #TEMP, PV := 6);   // CTU
   #TEMP := #CTU.Q;
END_REGION

REGION Network 3
   // 冷水机温度显示
   RUNG wire#powerrail
      #Modbus_Master.Modbus_Master(REQ := wire#w1, MB_ADDR := 1, MODE :=, DATA_ADDR := 40008, DATA_LEN := 1, DATA_PTR := #冷水温度读辅, DONE =>, BUSY =>, ERROR =>, STATUS =>)
      wire#w2
      { S7_Templates := "[SrcType := Int, DestType := Real]" } Convert(in := #冷水温度读辅, out => #ST1)
   END_RUNG
   RUNG wire#powerrail
      { S7_Templates := "SrcType := Int" } EQ_Contact(in1 := #CTU.CV, in2 := 0)
      P_Trig( #TP[0] )
   END_RUNG wire#w1
   RUNG wire#w2
      Div(in1 := #ST1, in2 := 10.0, out => #冷水温度读)
   END_RUNG
   // the same network as SCL:
   #_w1 := #CTU.CV = 0;
   #_w2 := #_w1 AND NOT #TP[0];   // rising edge
   #TP[0] := #_w1;
   #Modbus_Master(REQ := #_w2,   // Modbus_Master
                  MB_ADDR := 1,
                  DATA_ADDR := 40008,
                  DATA_LEN := 1,
                  DATA_PTR := #冷水温度读辅,
                  ENO => #_w3);
   IF #_w3 THEN
       #ST1 := INT_TO_REAL(#冷水温度读辅);
       #冷水温度读 := #ST1 / 10.0;
   END_IF;
END_REGION

REGION Network 4
   // 冷水机温度设定
   RUNG wire#powerrail
      #Modbus_Master.Modbus_Master(REQ := wire#w1, MB_ADDR := 1, MODE := 1, DATA_ADDR := 41026, DATA_LEN := 1, DATA_PTR := #冷水温度写辅, DONE =>, BUSY =>, ERROR =>, STATUS =>)
   END_RUNG
   RUNG wire#powerrail
      { S7_Templates := "SrcType := Int" } EQ_Contact(in1 := #CTU.CV, in2 := 1)
      P_Trig( #TP[1] )
   END_RUNG wire#w1
   RUNG wire#powerrail
      Contact( "AlwaysTRUE" )
      wire#w2
      Mul(in1 := #冷水温度写, in2 := 10.0, out => #ST16)
   END_RUNG
   RUNG wire#w2
      { S7_Templates := "[SrcType := Real, DestType := Int]" } Convert(in := #ST16, out => #冷水温度写辅)
   END_RUNG
   // the same network as SCL:
   #_w1 := #CTU.CV = 1;
   #_w2 := #_w1 AND NOT #TP[1];   // rising edge
   #TP[1] := #_w1;
   #Modbus_Master(REQ := #_w2, MB_ADDR := 1, MODE := 1, DATA_ADDR := 41026, DATA_LEN := 1, DATA_PTR := #冷水温度写辅);   // Modbus_Master
   IF "AlwaysTRUE" THEN
       #ST16 := #冷水温度写 * 10.0;
       #冷水温度写辅 := REAL_TO_INT(#ST16);
   END_IF;
END_REGION

REGION Network 5
   // 冷水机启停，11100，关，11110开
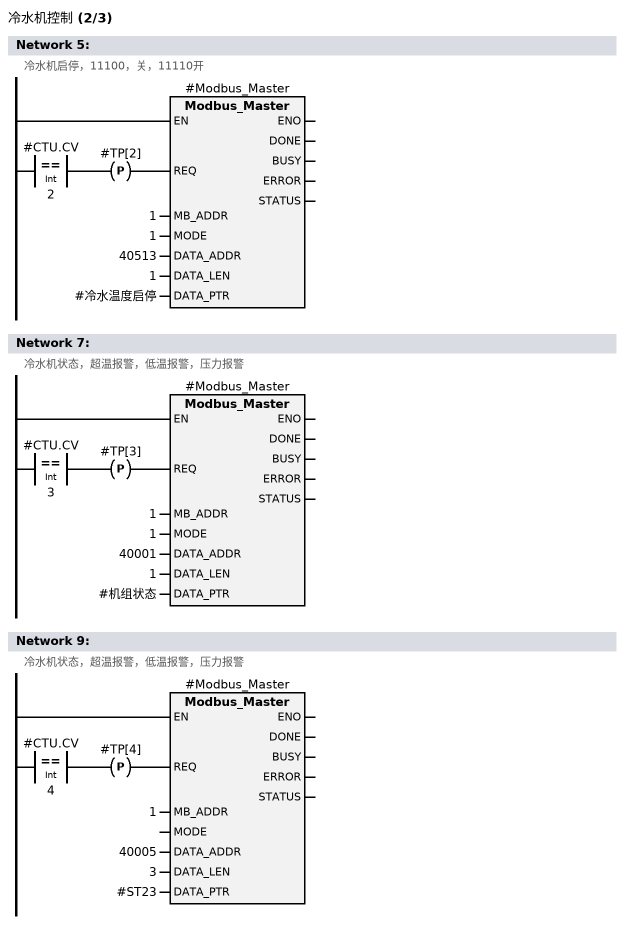
   RUNG wire#powerrail
      #Modbus_Master.Modbus_Master(REQ := wire#w1, MB_ADDR := 1, MODE := 1, DATA_ADDR := 40513, DATA_LEN := 1, DATA_PTR := #冷水温度启停, DONE =>, BUSY =>, ERROR =>, STATUS =>)
   END_RUNG
   RUNG wire#powerrail
      { S7_Templates := "SrcType := Int" } EQ_Contact(in1 := #CTU.CV, in2 := 2)
      P_Trig( #TP[2] )
   END_RUNG wire#w1
   // the same network as SCL:
   #_w1 := #CTU.CV = 2;
   #_w2 := #_w1 AND NOT #TP[2];   // rising edge
   #TP[2] := #_w1;
   #Modbus_Master(REQ := #_w2, MB_ADDR := 1, MODE := 1, DATA_ADDR := 40513, DATA_LEN := 1, DATA_PTR := #冷水温度启停);   // Modbus_Master
END_REGION

REGION Network 6 (SCL)
   IF #冷水启停开关 = TRUE THEN
       #冷水温度启停 := 114;

   END_IF;

   IF #冷水启停开关 = FALSE THEN
       #冷水温度启停 := 112;

   END_IF;
END_REGION

REGION Network 7
   // 冷水机状态，超温报警，低温报警，压力报警
   RUNG wire#powerrail
      #Modbus_Master.Modbus_Master(REQ := wire#w1, MB_ADDR := 1, MODE := 1, DATA_ADDR := 40001, DATA_LEN := 1, DATA_PTR := #机组状态, DONE =>, BUSY =>, ERROR =>, STATUS =>)
   END_RUNG
   RUNG wire#powerrail
      { S7_Templates := "SrcType := Int" } EQ_Contact(in1 := #CTU.CV, in2 := 3)
      P_Trig( #TP[3] )
   END_RUNG wire#w1
   // the same network as SCL:
   #_w1 := #CTU.CV = 3;
   #_w2 := #_w1 AND NOT #TP[3];   // rising edge
   #TP[3] := #_w1;
   #Modbus_Master(REQ := #_w2, MB_ADDR := 1, MODE := 1, DATA_ADDR := 40001, DATA_LEN := 1, DATA_PTR := #机组状态);   // Modbus_Master
END_REGION

REGION Network 9
   // 冷水机状态，超温报警，低温报警，压力报警
   RUNG wire#powerrail
      #Modbus_Master.Modbus_Master(REQ := wire#w1, MB_ADDR := 1, MODE :=, DATA_ADDR := 40005, DATA_LEN := 3, DATA_PTR := #ST23, DONE =>, BUSY =>, ERROR =>, STATUS =>)
   END_RUNG
   RUNG wire#powerrail
      { S7_Templates := "SrcType := Int" } EQ_Contact(in1 := #CTU.CV, in2 := 4)
      P_Trig( #TP[4] )
   END_RUNG wire#w1
   // the same network as SCL:
   #_w1 := #CTU.CV = 4;
   #_w2 := #_w1 AND NOT #TP[4];   // rising edge
   #TP[4] := #_w1;
   #Modbus_Master(REQ := #_w2, MB_ADDR := 1, DATA_ADDR := 40005, DATA_LEN := 3, DATA_PTR := #ST23);   // Modbus_Master
END_REGION

REGION Network 10 (SCL)
   IF #ST23[0]>0 OR #ST23[1]>0 OR #ST23[2]>0 THEN
       #冷水报警 := 1;
   ELSE
       #冷水报警 :=0;
   END_IF;
END_REGION

REGION Network 11
   // 冷水机温du
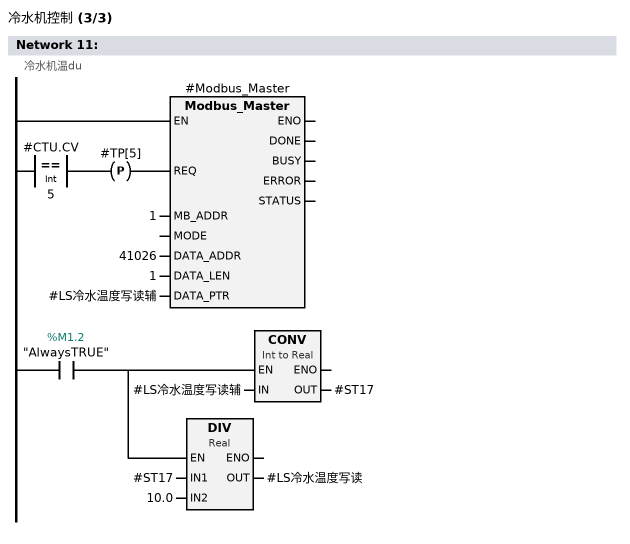
   RUNG wire#powerrail
      #Modbus_Master.Modbus_Master(REQ := wire#w1, MB_ADDR := 1, MODE :=, DATA_ADDR := 41026, DATA_LEN := 1, DATA_PTR := #LS冷水温度写读辅, DONE =>, BUSY =>, ERROR =>, STATUS =>)
   END_RUNG
   RUNG wire#powerrail
      { S7_Templates := "SrcType := Int" } EQ_Contact(in1 := #CTU.CV, in2 := 5)
      P_Trig( #TP[5] )
   END_RUNG wire#w1
   RUNG wire#powerrail
      Contact( "AlwaysTRUE" )
      wire#w2
      { S7_Templates := "[SrcType := Int, DestType := Real]" } Convert(in := #LS冷水温度写读辅, out => #ST17)
   END_RUNG
   RUNG wire#w2
      { S7_Templates := "SrcType := Real" } Div(in1 := #ST17, in2 := 10.0, out => #LS冷水温度写读)
   END_RUNG
   // the same network as SCL:
   #_w1 := #CTU.CV = 5;
   #_w2 := #_w1 AND NOT #TP[5];   // rising edge
   #TP[5] := #_w1;
   #Modbus_Master(REQ := #_w2, MB_ADDR := 1, DATA_ADDR := 41026, DATA_LEN := 1, DATA_PTR := #LS冷水温度写读辅);   // Modbus_Master
   IF "AlwaysTRUE" THEN
       #ST17 := INT_TO_REAL(#LS冷水温度写读辅);
       #LS冷水温度写读 := #ST17 / 10.0;
   END_IF;
END_REGION
END_FUNCTION_BLOCK

FUNCTION_BLOCK "油炉控制"   // FB52, LAD
{ S7_Optimized_Access := 'FALSE' }
VERSION : 0.1
// stored: AutoNumber true, IsIECCheckEnabled false, SetENOAutomatically false, UDAEnableTagReadback false
   VAR_IN_OUT
      油炉温度写 : Real;
      油炉温度读 : Real;
      油炉循环泵启停 : Bool;
      油炉报警 : Bool;
      油炉冷却阀启停状态 : Bool;
      油炉加热泵启停状态 : Bool;
      油炉加热器1状态 : Bool;
      油炉加热器2状态 : Bool;
      油炉运行状态 : Bool;
      油炉自整定状态 : Bool;
      油炉强制冷却状态 : Bool;
      YL油炉温度写读 : Real;
   END_VAR
   VAR DB_SPECIFIC
      CTU { S7_SetPoint := 'True'} : CTU_INT;
      TEMP { S7_SetPoint := 'True'} : Bool;
      TP : Array[0..40] of Bool;
      油炉温度读辅 : Int;
      油炉温度写辅 : Int;
      ST1 : Real;
      ST2 : Real;
      ST3 : Real;
      ST4 : Real;
      ST5 : Real;
      ST16 : Real;
      ST17 : Real;
      ST18 : Real;
      ST20 : Real;
      ST21 : Real;
      ST22 : Real;
      油炉状态1 : Int;
      油炉状态2 : Int;
      油炉启停字 : Int;
      油炉加热状态 : Int;
      油炉运行标志 : Int;
      YL油炉温度写读辅 : Int;
   END_VAR
   VAR
      Modbus_Comm_Load { S7_SetPoint := 'True'} : Modbus_Comm_Load;
      Modbus_Master { S7_SetPoint := 'True'} : Modbus_Master;
   END_VAR
   VAR_TEMP   // added for the SCL form of the ladder/FBD networks
      _w1 : Bool;
      _w2 : Bool;
      _w3 : Bool;
   END_VAR
BEGIN

REGION Network 1
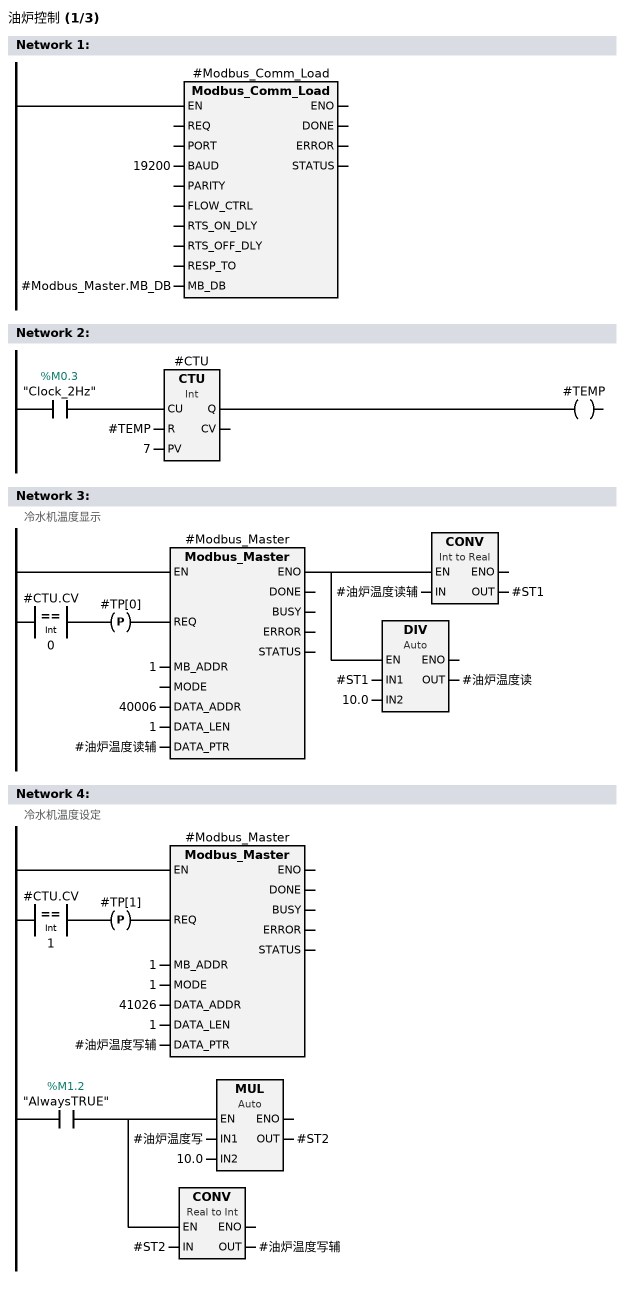
   RUNG wire#powerrail
      #Modbus_Comm_Load.Modbus_Comm_Load(REQ :=, PORT :=, BAUD := 19200, PARITY :=, FLOW_CTRL :=, RTS_ON_DLY :=, RTS_OFF_DLY :=, RESP_TO :=, MB_DB := #Modbus_Master.MB_DB, DONE =>, ERROR =>, STATUS =>)
   END_RUNG
   // the same network as SCL:
   #Modbus_Comm_Load(BAUD := 19200, MB_DB := #Modbus_Master.MB_DB);   // Modbus_Comm_Load
END_REGION

REGION Network 2
   RUNG wire#powerrail
      Contact( "Clock_2Hz" )
      { S7_Templates := "value_type := Int" } #CTU.CTU(r := #TEMP, pv := 7, cv =>)
      Coil( #TEMP )
   END_RUNG
   // the same network as SCL:
   #CTU(CU := "Clock_2Hz", R := #TEMP, PV := 7);   // CTU
   #TEMP := #CTU.Q;
END_REGION

REGION Network 3
   // 冷水机温度显示
   RUNG wire#powerrail
      #Modbus_Master.Modbus_Master(REQ := wire#w1, MB_ADDR := 1, MODE :=, DATA_ADDR := 40006, DATA_LEN := 1, DATA_PTR := #油炉温度读辅, DONE =>, BUSY =>, ERROR =>, STATUS =>)
      wire#w2
      { S7_Templates := "[SrcType := Int, DestType := Real]" } Convert(in := #油炉温度读辅, out => #ST1)
   END_RUNG
   RUNG wire#powerrail
      { S7_Templates := "SrcType := Int" } EQ_Contact(in1 := #CTU.CV, in2 := 0)
      P_Trig( #TP[0] )
   END_RUNG wire#w1
   RUNG wire#w2
      Div(in1 := #ST1, in2 := 10.0, out => #油炉温度读)
   END_RUNG
   // the same network as SCL:
   #_w1 := #CTU.CV = 0;
   #_w2 := #_w1 AND NOT #TP[0];   // rising edge
   #TP[0] := #_w1;
   #Modbus_Master(REQ := #_w2,   // Modbus_Master
                  MB_ADDR := 1,
                  DATA_ADDR := 40006,
                  DATA_LEN := 1,
                  DATA_PTR := #油炉温度读辅,
                  ENO => #_w3);
   IF #_w3 THEN
       #ST1 := INT_TO_REAL(#油炉温度读辅);
       #油炉温度读 := #ST1 / 10.0;
   END_IF;
END_REGION

REGION Network 4
   // 冷水机温度设定
   RUNG wire#powerrail
      #Modbus_Master.Modbus_Master(REQ := wire#w1, MB_ADDR := 1, MODE := 1, DATA_ADDR := 41026, DATA_LEN := 1, DATA_PTR := #油炉温度写辅, DONE =>, BUSY =>, ERROR =>, STATUS =>)
   END_RUNG
   RUNG wire#powerrail
      { S7_Templates := "SrcType := Int" } EQ_Contact(in1 := #CTU.CV, in2 := 1)
      P_Trig( #TP[1] )
   END_RUNG wire#w1
   RUNG wire#powerrail
      Contact( "AlwaysTRUE" )
      wire#w2
      Mul(in1 := #油炉温度写, in2 := 10.0, out => #ST2)
   END_RUNG
   RUNG wire#w2
      { S7_Templates := "[SrcType := Real, DestType := Int]" } Convert(in := #ST2, out => #油炉温度写辅)
   END_RUNG
   // the same network as SCL:
   #_w1 := #CTU.CV = 1;
   #_w2 := #_w1 AND NOT #TP[1];   // rising edge
   #TP[1] := #_w1;
   #Modbus_Master(REQ := #_w2, MB_ADDR := 1, MODE := 1, DATA_ADDR := 41026, DATA_LEN := 1, DATA_PTR := #油炉温度写辅);   // Modbus_Master
   IF "AlwaysTRUE" THEN
       #ST2 := #油炉温度写 * 10.0;
       #油炉温度写辅 := REAL_TO_INT(#ST2);
   END_IF;
END_REGION

REGION Network 5
   // 冷水机温度设定
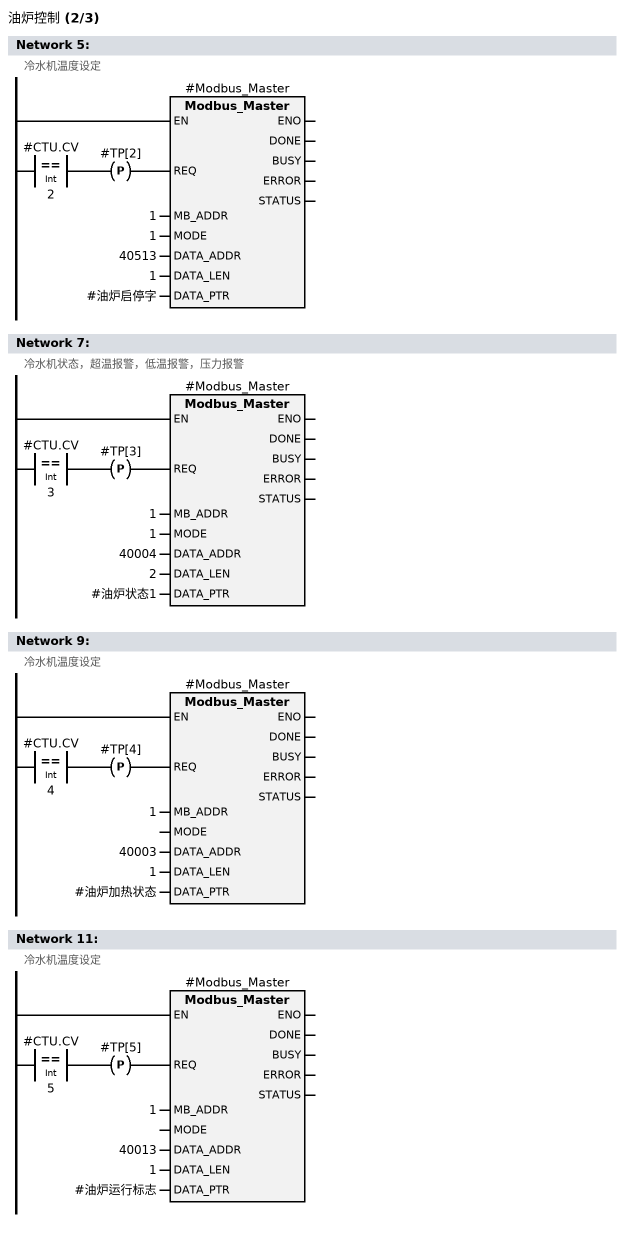
   RUNG wire#powerrail
      #Modbus_Master.Modbus_Master(REQ := wire#w1, MB_ADDR := 1, MODE := 1, DATA_ADDR := 40513, DATA_LEN := 1, DATA_PTR := #油炉启停字, DONE =>, BUSY =>, ERROR =>, STATUS =>)
   END_RUNG
   RUNG wire#powerrail
      { S7_Templates := "SrcType := Int" } EQ_Contact(in1 := #CTU.CV, in2 := 2)
      P_Trig( #TP[2] )
   END_RUNG wire#w1
   // the same network as SCL:
   #_w1 := #CTU.CV = 2;
   #_w2 := #_w1 AND NOT #TP[2];   // rising edge
   #TP[2] := #_w1;
   #Modbus_Master(REQ := #_w2, MB_ADDR := 1, MODE := 1, DATA_ADDR := 40513, DATA_LEN := 1, DATA_PTR := #油炉启停字);   // Modbus_Master
END_REGION

REGION Network 6 (SCL)
   IF #油炉循环泵启停 = TRUE THEN
       #油炉启停字:= 114;
   ELSE
       #油炉启停字 := 112;
   END_IF;
END_REGION

REGION Network 7
   // 冷水机状态，超温报警，低温报警，压力报警
   RUNG wire#powerrail
      #Modbus_Master.Modbus_Master(REQ := wire#w1, MB_ADDR := 1, MODE := 1, DATA_ADDR := 40004, DATA_LEN := 2, DATA_PTR := #油炉状态1, DONE =>, BUSY =>, ERROR =>, STATUS =>)
   END_RUNG
   RUNG wire#powerrail
      { S7_Templates := "SrcType := Int" } EQ_Contact(in1 := #CTU.CV, in2 := 3)
      P_Trig( #TP[3] )
   END_RUNG wire#w1
   // the same network as SCL:
   #_w1 := #CTU.CV = 3;
   #_w2 := #_w1 AND NOT #TP[3];   // rising edge
   #TP[3] := #_w1;
   #Modbus_Master(REQ := #_w2, MB_ADDR := 1, MODE := 1, DATA_ADDR := 40004, DATA_LEN := 2, DATA_PTR := #油炉状态1);   // Modbus_Master
END_REGION

REGION Network 8 (SCL)
   IF #油炉状态1>1 OR #油炉状态2>1 THEN
       #油炉报警 := TRUE;
   ELSE
       #油炉报警 := FALSE;
   END_IF;
END_REGION

REGION Network 9
   // 冷水机温度设定
   RUNG wire#powerrail
      #Modbus_Master.Modbus_Master(REQ := wire#w1, MB_ADDR := 1, MODE :=, DATA_ADDR := 40003, DATA_LEN := 1, DATA_PTR := #油炉加热状态, DONE =>, BUSY =>, ERROR =>, STATUS =>)
   END_RUNG
   RUNG wire#powerrail
      { S7_Templates := "SrcType := Int" } EQ_Contact(in1 := #CTU.CV, in2 := 4)
      P_Trig( #TP[4] )
   END_RUNG wire#w1
   // the same network as SCL:
   #_w1 := #CTU.CV = 4;
   #_w2 := #_w1 AND NOT #TP[4];   // rising edge
   #TP[4] := #_w1;
   #Modbus_Master(REQ := #_w2, MB_ADDR := 1, DATA_ADDR := 40003, DATA_LEN := 1, DATA_PTR := #油炉加热状态);   // Modbus_Master
END_REGION

REGION Network 10 (SCL)
   IF #油炉加热状态 >= 8 THEN
       #油炉冷却阀启停状态 := TRUE;
   ELSE
       #油炉冷却阀启停状态 := FALSE;
   END_IF;

   IF #油炉加热状态 >= 4 THEN
       #油炉加热泵启停状态 := TRUE;
   ELSE
       #油炉加热泵启停状态 := FALSE;
   END_IF;


   IF #油炉加热状态 >= 2 THEN
       #油炉加热器2状态 := TRUE;
   ELSE
       #油炉加热器2状态 := FALSE;
   END_IF;

   IF #油炉加热状态 >= 1 THEN
       #油炉加热器1状态 := TRUE;
   ELSE
       #油炉加热器1状态 := FALSE;
   END_IF;
END_REGION

REGION Network 11
   // 冷水机温度设定
   RUNG wire#powerrail
      #Modbus_Master.Modbus_Master(REQ := wire#w1, MB_ADDR := 1, MODE :=, DATA_ADDR := 40013, DATA_LEN := 1, DATA_PTR := #油炉运行标志, DONE =>, BUSY =>, ERROR =>, STATUS =>)
   END_RUNG
   RUNG wire#powerrail
      { S7_Templates := "SrcType := Int" } EQ_Contact(in1 := #CTU.CV, in2 := 5)
      P_Trig( #TP[5] )
   END_RUNG wire#w1
   // the same network as SCL:
   #_w1 := #CTU.CV = 5;
   #_w2 := #_w1 AND NOT #TP[5];   // rising edge
   #TP[5] := #_w1;
   #Modbus_Master(REQ := #_w2, MB_ADDR := 1, DATA_ADDR := 40013, DATA_LEN := 1, DATA_PTR := #油炉运行标志);   // Modbus_Master
END_REGION

REGION Network 12
   // 冷水机温du
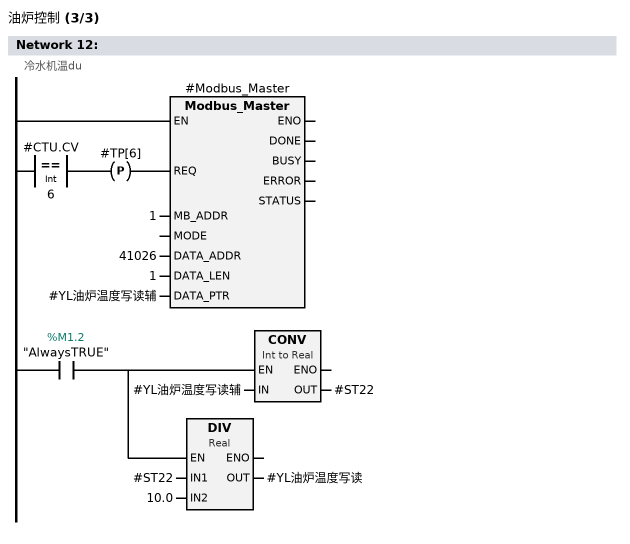
   RUNG wire#powerrail
      #Modbus_Master.Modbus_Master(REQ := wire#w1, MB_ADDR := 1, MODE :=, DATA_ADDR := 41026, DATA_LEN := 1, DATA_PTR := #YL油炉温度写读辅, DONE =>, BUSY =>, ERROR =>, STATUS =>)
   END_RUNG
   RUNG wire#powerrail
      { S7_Templates := "SrcType := Int" } EQ_Contact(in1 := #CTU.CV, in2 := 6)
      P_Trig( #TP[6] )
   END_RUNG wire#w1
   RUNG wire#powerrail
      Contact( "AlwaysTRUE" )
      wire#w2
      { S7_Templates := "[SrcType := Int, DestType := Real]" } Convert(in := #YL油炉温度写读辅, out => #ST22)
   END_RUNG
   RUNG wire#w2
      { S7_Templates := "SrcType := Real" } Div(in1 := #ST22, in2 := 10.0, out => #YL油炉温度写读)
   END_RUNG
   // the same network as SCL:
   #_w1 := #CTU.CV = 6;
   #_w2 := #_w1 AND NOT #TP[6];   // rising edge
   #TP[6] := #_w1;
   #Modbus_Master(REQ := #_w2, MB_ADDR := 1, DATA_ADDR := 41026, DATA_LEN := 1, DATA_PTR := #YL油炉温度写读辅);   // Modbus_Master
   IF "AlwaysTRUE" THEN
       #ST22 := INT_TO_REAL(#YL油炉温度写读辅);
       #YL油炉温度写读 := #ST22 / 10.0;
   END_IF;
END_REGION

REGION Network 13 (SCL)
   IF #油炉运行标志 >= 4 THEN
       #油炉强制冷却状态 := TRUE;
   ELSE
       #油炉强制冷却状态 := FALSE;
   END_IF;

   IF #油炉运行标志 >= 2 THEN
       #油炉自整定状态 := TRUE;
   ELSE
       #油炉自整定状态 := FALSE;
   END_IF;


   IF #油炉运行标志 >= 1 THEN
       #油炉运行状态 := TRUE;
   ELSE
       #油炉运行状态 := FALSE;
   END_IF;
END_REGION
END_FUNCTION_BLOCK

FUNCTION_BLOCK "称重与流量"   // FB57, LAD
{ S7_Optimized_Access := 'FALSE' }
VERSION : 0.1
// stored: AutoNumber true, IsIECCheckEnabled false, SetENOAutomatically false, UDAEnableTagReadback false
   VAR_OUTPUT
      A瞬时流量 : Real;
      A瞬时流量AT AT A瞬时流量 : Array[0..1] of Word;
      A瞬时流速 : Real;
      A瞬时流速AT AT A瞬时流速 : Array[0..1] of Word;
      A当前电流 : Real;
      A当前电流AT AT A当前电流 : Array[0..1] of Word;
      A介质温度 : Real;
      A介质温度AT AT A介质温度 : Array[0..1] of Word;
      A当前采集 : Real;
      A当前采集AT AT A当前采集 : Array[0..1] of Word;
      A流速下限 : Real;
      A流速下限AT AT A流速下限 : Array[0..1] of Word;
      A流速上限 : Real;
      A流速上限AT AT A流速上限 : Array[0..1] of Word;
      A管道内径 : Real;
      A管道内径AT AT A管道内径 : Array[0..1] of Word;
      B瞬时流量 : Real;
      B瞬时流量AT AT B瞬时流量 : Array[0..1] of Word;
      B瞬时流速 : Real;
      B瞬时流速AT AT B瞬时流速 : Array[0..1] of Word;
      B当前电流 : Real;
      B当前电流AT AT B当前电流 : Array[0..1] of Word;
      B介质温度 : Real;
      B介质温度AT AT B介质温度 : Array[0..1] of Word;
      B当前采集 : Real;
      B当前采集AT AT B当前采集 : Array[0..1] of Word;
      B流速下限 : Real;
      B流速下限AT AT B流速下限 : Array[0..1] of Word;
      B流速上限 : Real;
      B流速上限AT AT B流速上限 : Array[0..1] of Word;
      B管道内径 : Real;
      B管道内径AT AT B管道内径 : Array[0..1] of Word;
   END_VAR
   VAR_IN_OUT
      "秤操作-去皮" : Bool;
      读重量 : Real;
   END_VAR
   VAR DB_SPECIFIC
      CTU { S7_SetPoint := 'True'} : CTU_INT;
      TEMP { S7_SetPoint := 'True'} : Bool;
      TON1 : TON_TIME;
      TP : Array[0..40] of Bool;
      秤操作辅助 : Int;
      CZTFZ : Int;
   END_VAR
   VAR
      CZT AT CZTFZ : Array[0..15] of Bool;
   END_VAR
   VAR DB_SPECIFIC
      ST1 : Array[0..5] of Word;
      ST2 : Array[0..7] of Word;
      ST3 : Array[0..1] of Word;
      ST4 : Array[0..5] of Word;
      ST5 : Array[0..7] of Word;
      ST6 : Array[0..1] of Word;
      ST7 : Array[0..1] of Word;
      读重量辅助 : DInt;
   END_VAR
   VAR
      读重量辅助AT AT 读重量辅助 : Array[0..1] of Word;
      Modbus_Comm_Load { S7_SetPoint := 'True'} : Modbus_Comm_Load;
      Modbus_Master { S7_SetPoint := 'True'} : Modbus_Master;
   END_VAR
   VAR_TEMP   // added for the SCL form of the ladder/FBD networks
      _w1 : Bool;
      _w2 : Bool;
      _w3 : Bool;
   END_VAR
BEGIN

REGION Network 1
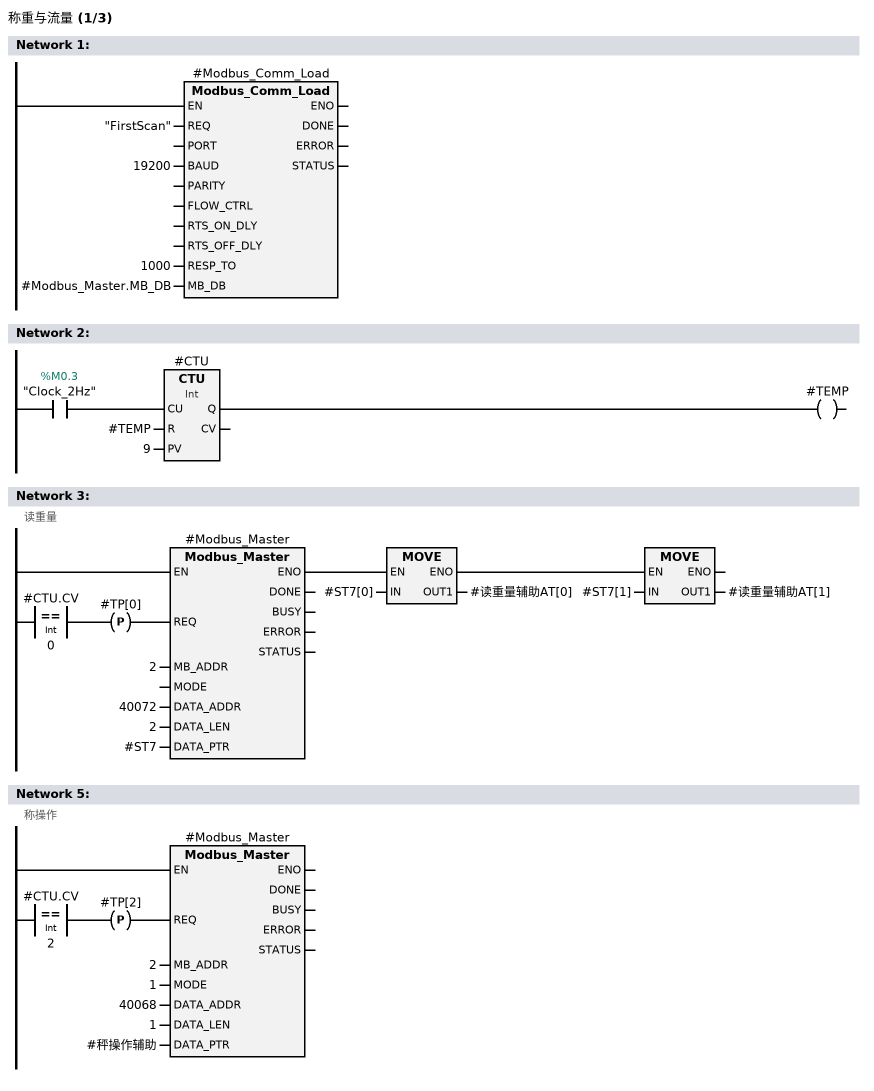
   RUNG wire#powerrail
      #Modbus_Comm_Load.Modbus_Comm_Load(REQ := "FirstScan", PORT :=, BAUD := 19200, PARITY :=, FLOW_CTRL :=, RTS_ON_DLY :=, RTS_OFF_DLY :=, RESP_TO := 1000, MB_DB := #Modbus_Master.MB_DB, DONE =>, ERROR =>, STATUS =>)
   END_RUNG
   // the same network as SCL:
   #Modbus_Comm_Load(REQ := "FirstScan", BAUD := 19200, RESP_TO := 1000, MB_DB := #Modbus_Master.MB_DB);   // Modbus_Comm_Load
END_REGION

REGION Network 2
   RUNG wire#powerrail
      Contact( "Clock_2Hz" )
      { S7_Templates := "value_type := Int" } #CTU.CTU(r := #TEMP, pv := 9, cv =>)
      Coil( #TEMP )
   END_RUNG
   // the same network as SCL:
   #CTU(CU := "Clock_2Hz", R := #TEMP, PV := 9);   // CTU
   #TEMP := #CTU.Q;
END_REGION

REGION Network 3
   // 读重量
   RUNG wire#powerrail
      #Modbus_Master.Modbus_Master(REQ := wire#w1, MB_ADDR := 2, MODE :=, DATA_ADDR := 40072, DATA_LEN := 2, DATA_PTR := #ST7, DONE =>, BUSY =>, ERROR =>, STATUS =>)
      Move(in := #ST7[0], out1 => #读重量辅助AT[0])
      Move(in := #ST7[1], out1 => #读重量辅助AT[1])
   END_RUNG
   RUNG wire#powerrail
      { S7_Templates := "SrcType := Int" } EQ_Contact(in1 := #CTU.CV, in2 := 0)
      P_Trig( #TP[0] )
   END_RUNG wire#w1
   // the same network as SCL:
   #_w1 := #CTU.CV = 0;
   #_w2 := #_w1 AND NOT #TP[0];   // rising edge
   #TP[0] := #_w1;
   #Modbus_Master(REQ := #_w2, MB_ADDR := 2, DATA_ADDR := 40072, DATA_LEN := 2, DATA_PTR := #ST7, ENO => #_w3);   // Modbus_Master
   IF #_w3 THEN
       #读重量辅助AT[0] := #ST7[0];
       #读重量辅助AT[1] := #ST7[1];
   END_IF;
END_REGION

REGION Network 4 (SCL)


   #读重量 := DINT_TO_REAL(#读重量辅助) * 0.01;
END_REGION

REGION Network 5
   // 称操作
   RUNG wire#powerrail
      #Modbus_Master.Modbus_Master(REQ := wire#w1, MB_ADDR := 2, MODE := 1, DATA_ADDR := 40068, DATA_LEN := 1, DATA_PTR := #秤操作辅助, DONE =>, BUSY =>, ERROR =>, STATUS =>)
   END_RUNG
   RUNG wire#powerrail
      { S7_Templates := "SrcType := Int" } EQ_Contact(in1 := #CTU.CV, in2 := 2)
      P_Trig( #TP[2] )
   END_RUNG wire#w1
   // the same network as SCL:
   #_w1 := #CTU.CV = 2;
   #_w2 := #_w1 AND NOT #TP[2];   // rising edge
   #TP[2] := #_w1;
   #Modbus_Master(REQ := #_w2, MB_ADDR := 2, MODE := 1, DATA_ADDR := 40068, DATA_LEN := 1, DATA_PTR := #秤操作辅助);   // Modbus_Master
END_REGION

REGION Network 6 (SCL)


   IF #"秤操作-去皮" = TRUE THEN
       #秤操作辅助 := 11;
       #"秤操作-去皮" := 0;

   END_IF;



   #TON1(IN := #秤操作辅助<>0,
         PT := T#5S);

   IF #TON1.Q THEN
       #秤操作辅助 := 0;

   END_IF;
END_REGION

REGION Network 7
   // 读流量
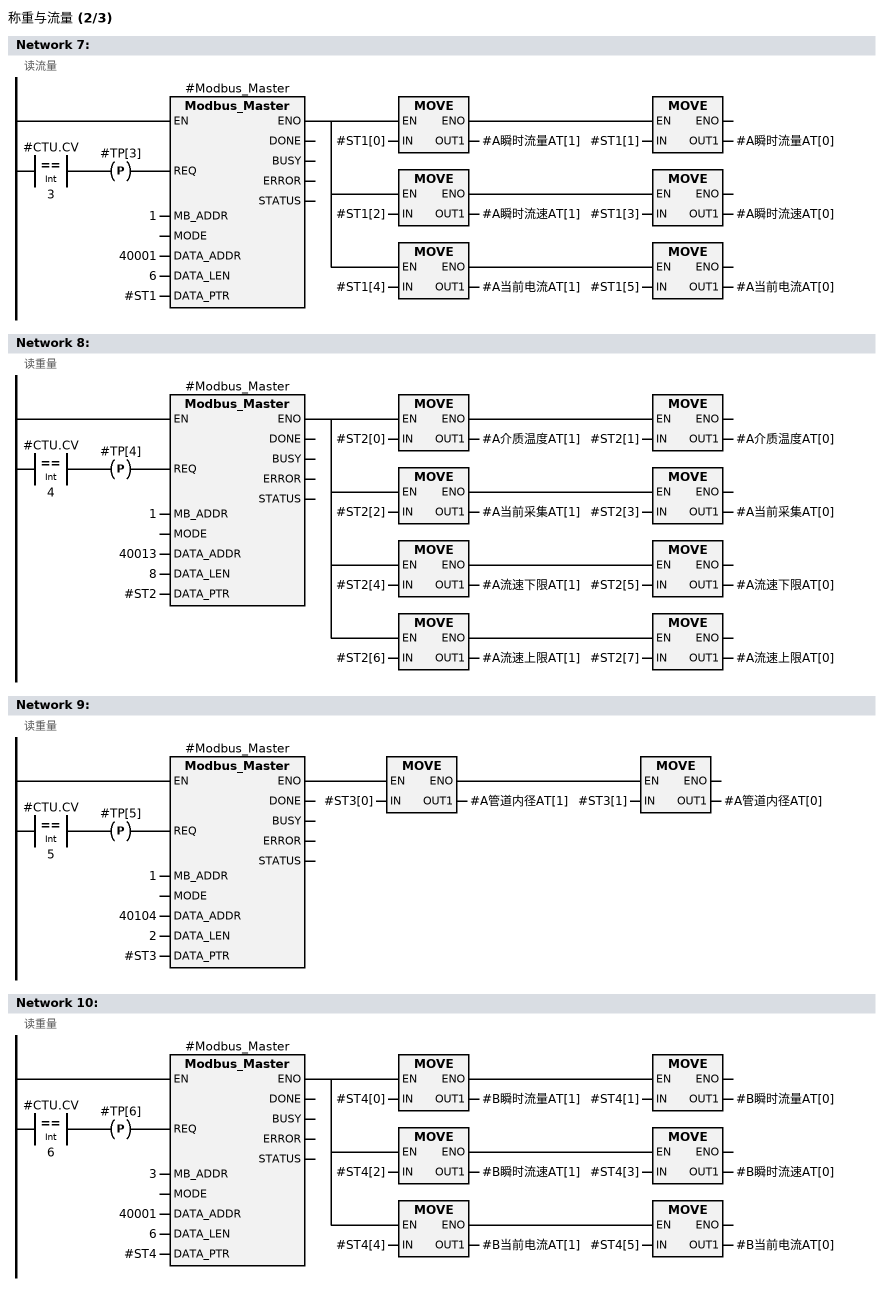
   RUNG wire#powerrail
      #Modbus_Master.Modbus_Master(REQ := wire#w1, MB_ADDR := 1, MODE :=, DATA_ADDR := 40001, DATA_LEN := 6, DATA_PTR := #ST1, DONE =>, BUSY =>, ERROR =>, STATUS =>)
      wire#w2
      Move(in := #ST1[0], out1 => #A瞬时流量AT[1])
      Move(in := #ST1[1], out1 => #A瞬时流量AT[0])
   END_RUNG
   RUNG wire#powerrail
      { S7_Templates := "SrcType := Int" } EQ_Contact(in1 := #CTU.CV, in2 := 3)
      P_Trig( #TP[3] )
   END_RUNG wire#w1
   RUNG wire#w2
      Move(in := #ST1[2], out1 => #A瞬时流速AT[1])
      Move(in := #ST1[3], out1 => #A瞬时流速AT[0])
   END_RUNG
   RUNG wire#w2
      Move(in := #ST1[4], out1 => #A当前电流AT[1])
      Move(in := #ST1[5], out1 => #A当前电流AT[0])
   END_RUNG
   // the same network as SCL:
   #_w1 := #CTU.CV = 3;
   #_w2 := #_w1 AND NOT #TP[3];   // rising edge
   #TP[3] := #_w1;
   #Modbus_Master(REQ := #_w2, MB_ADDR := 1, DATA_ADDR := 40001, DATA_LEN := 6, DATA_PTR := #ST1, ENO => #_w3);   // Modbus_Master
   IF #_w3 THEN
       #A瞬时流量AT[1] := #ST1[0];
       #A瞬时流量AT[0] := #ST1[1];
       #A瞬时流速AT[1] := #ST1[2];
       #A瞬时流速AT[0] := #ST1[3];
       #A当前电流AT[1] := #ST1[4];
       #A当前电流AT[0] := #ST1[5];
   END_IF;
END_REGION

REGION Network 8
   // 读重量
   RUNG wire#powerrail
      #Modbus_Master.Modbus_Master(REQ := wire#w1, MB_ADDR := 1, MODE :=, DATA_ADDR := 40013, DATA_LEN := 8, DATA_PTR := #ST2, DONE =>, BUSY =>, ERROR =>, STATUS =>)
      wire#w2
      Move(in := #ST2[0], out1 => #A介质温度AT[1])
      Move(in := #ST2[1], out1 => #A介质温度AT[0])
   END_RUNG
   RUNG wire#powerrail
      { S7_Templates := "SrcType := Int" } EQ_Contact(in1 := #CTU.CV, in2 := 4)
      P_Trig( #TP[4] )
   END_RUNG wire#w1
   RUNG wire#w2
      Move(in := #ST2[2], out1 => #A当前采集AT[1])
      Move(in := #ST2[3], out1 => #A当前采集AT[0])
   END_RUNG
   RUNG wire#w2
      Move(in := #ST2[4], out1 => #A流速下限AT[1])
      Move(in := #ST2[5], out1 => #A流速下限AT[0])
   END_RUNG
   RUNG wire#w2
      Move(in := #ST2[6], out1 => #A流速上限AT[1])
      Move(in := #ST2[7], out1 => #A流速上限AT[0])
   END_RUNG
   // the same network as SCL:
   #_w1 := #CTU.CV = 4;
   #_w2 := #_w1 AND NOT #TP[4];   // rising edge
   #TP[4] := #_w1;
   #Modbus_Master(REQ := #_w2, MB_ADDR := 1, DATA_ADDR := 40013, DATA_LEN := 8, DATA_PTR := #ST2, ENO => #_w3);   // Modbus_Master
   IF #_w3 THEN
       #A介质温度AT[1] := #ST2[0];
       #A介质温度AT[0] := #ST2[1];
       #A当前采集AT[1] := #ST2[2];
       #A当前采集AT[0] := #ST2[3];
       #A流速下限AT[1] := #ST2[4];
       #A流速下限AT[0] := #ST2[5];
       #A流速上限AT[1] := #ST2[6];
       #A流速上限AT[0] := #ST2[7];
   END_IF;
END_REGION

REGION Network 9
   // 读重量
   RUNG wire#powerrail
      #Modbus_Master.Modbus_Master(REQ := wire#w1, MB_ADDR := 1, MODE :=, DATA_ADDR := 40104, DATA_LEN := 2, DATA_PTR := #ST3, DONE =>, BUSY =>, ERROR =>, STATUS =>)
      Move(in := #ST3[0], out1 => #A管道内径AT[1])
      Move(in := #ST3[1], out1 => #A管道内径AT[0])
   END_RUNG
   RUNG wire#powerrail
      { S7_Templates := "SrcType := Int" } EQ_Contact(in1 := #CTU.CV, in2 := 5)
      P_Trig( #TP[5] )
   END_RUNG wire#w1
   // the same network as SCL:
   #_w1 := #CTU.CV = 5;
   #_w2 := #_w1 AND NOT #TP[5];   // rising edge
   #TP[5] := #_w1;
   #Modbus_Master(REQ := #_w2, MB_ADDR := 1, DATA_ADDR := 40104, DATA_LEN := 2, DATA_PTR := #ST3, ENO => #_w3);   // Modbus_Master
   IF #_w3 THEN
       #A管道内径AT[1] := #ST3[0];
       #A管道内径AT[0] := #ST3[1];
   END_IF;
END_REGION

REGION Network 10
   // 读重量
   RUNG wire#powerrail
      #Modbus_Master.Modbus_Master(REQ := wire#w1, MB_ADDR := 3, MODE :=, DATA_ADDR := 40001, DATA_LEN := 6, DATA_PTR := #ST4, DONE =>, BUSY =>, ERROR =>, STATUS =>)
      wire#w2
      Move(in := #ST4[0], out1 => #B瞬时流量AT[1])
      Move(in := #ST4[1], out1 => #B瞬时流量AT[0])
   END_RUNG
   RUNG wire#powerrail
      { S7_Templates := "SrcType := Int" } EQ_Contact(in1 := #CTU.CV, in2 := 6)
      P_Trig( #TP[6] )
   END_RUNG wire#w1
   RUNG wire#w2
      Move(in := #ST4[2], out1 => #B瞬时流速AT[1])
      Move(in := #ST4[3], out1 => #B瞬时流速AT[0])
   END_RUNG
   RUNG wire#w2
      Move(in := #ST4[4], out1 => #B当前电流AT[1])
      Move(in := #ST4[5], out1 => #B当前电流AT[0])
   END_RUNG
   // the same network as SCL:
   #_w1 := #CTU.CV = 6;
   #_w2 := #_w1 AND NOT #TP[6];   // rising edge
   #TP[6] := #_w1;
   #Modbus_Master(REQ := #_w2, MB_ADDR := 3, DATA_ADDR := 40001, DATA_LEN := 6, DATA_PTR := #ST4, ENO => #_w3);   // Modbus_Master
   IF #_w3 THEN
       #B瞬时流量AT[1] := #ST4[0];
       #B瞬时流量AT[0] := #ST4[1];
       #B瞬时流速AT[1] := #ST4[2];
       #B瞬时流速AT[0] := #ST4[3];
       #B当前电流AT[1] := #ST4[4];
       #B当前电流AT[0] := #ST4[5];
   END_IF;
END_REGION

REGION Network 11
   // 读重量
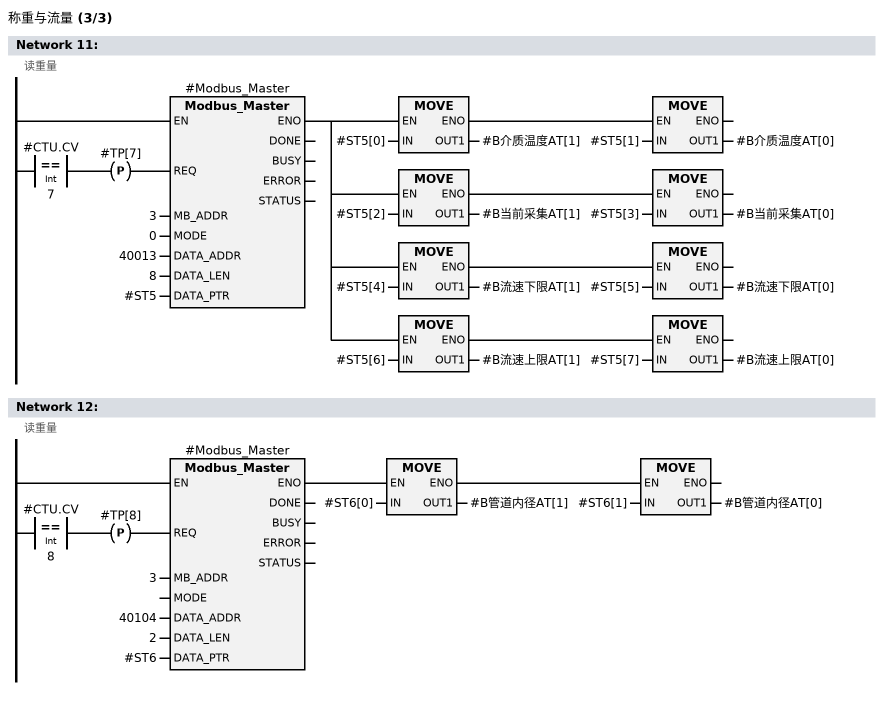
   RUNG wire#powerrail
      #Modbus_Master.Modbus_Master(REQ := wire#w1, MB_ADDR := 3, MODE := 0, DATA_ADDR := 40013, DATA_LEN := 8, DATA_PTR := #ST5, DONE =>, BUSY =>, ERROR =>, STATUS =>)
      wire#w2
      Move(in := #ST5[0], out1 => #B介质温度AT[1])
      Move(in := #ST5[1], out1 => #B介质温度AT[0])
   END_RUNG
   RUNG wire#powerrail
      { S7_Templates := "SrcType := Int" } EQ_Contact(in1 := #CTU.CV, in2 := 7)
      P_Trig( #TP[7] )
   END_RUNG wire#w1
   RUNG wire#w2
      Move(in := #ST5[2], out1 => #B当前采集AT[1])
      Move(in := #ST5[3], out1 => #B当前采集AT[0])
   END_RUNG
   RUNG wire#w2
      Move(in := #ST5[4], out1 => #B流速下限AT[1])
      Move(in := #ST5[5], out1 => #B流速下限AT[0])
   END_RUNG
   RUNG wire#w2
      Move(in := #ST5[6], out1 => #B流速上限AT[1])
      Move(in := #ST5[7], out1 => #B流速上限AT[0])
   END_RUNG
   // the same network as SCL:
   #_w1 := #CTU.CV = 7;
   #_w2 := #_w1 AND NOT #TP[7];   // rising edge
   #TP[7] := #_w1;
   #Modbus_Master(REQ := #_w2,   // Modbus_Master
                  MB_ADDR := 3,
                  MODE := 0,
                  DATA_ADDR := 40013,
                  DATA_LEN := 8,
                  DATA_PTR := #ST5,
                  ENO => #_w3);
   IF #_w3 THEN
       #B介质温度AT[1] := #ST5[0];
       #B介质温度AT[0] := #ST5[1];
       #B当前采集AT[1] := #ST5[2];
       #B当前采集AT[0] := #ST5[3];
       #B流速下限AT[1] := #ST5[4];
       #B流速下限AT[0] := #ST5[5];
       #B流速上限AT[1] := #ST5[6];
       #B流速上限AT[0] := #ST5[7];
   END_IF;
END_REGION

